LIN {X 0,Y 254.185,Z 743.005,A -85,B 0,C 180,E1 -18348.841,E2 -18348.841} C_VEL
LIN {X 0,Y 254.451,Z 743.746,A -85,B 0,C 180,E1 -18350.461,E2 -18350.461} C_VEL
LIN {X 0,Y 255.037,Z 744.003,A -85,B 0,C 180,E1 -18352.785,E2 -18352.785} C_VEL
LIN {X 0,Y 255.836,Z 743.277,A -85,B 0,C 180,E1 -18355.273,E2 -18355.273} C_VEL
LIN {X 0,Y 256.521,Z 742.248,A -85,B 0,C 180,E1 -18356.859,E2 -18356.859} C_VEL
LIN {X 0,Y 257.385,Z 740.801,A -85,B 0,C 180,E1 -18358.436,E2 -18358.436} C_VEL
LIN {X 0,Y 259.004,Z 737.791,A -85,B 0,C 180,E1 -18360.778,E2 -18360.778} C_VEL
LIN {X 0,Y 260.963,Z 733.697,A -85,B 0,C 180,E1 -18363.088,E2 -18363.088} C_VEL
LIN {X 0,Y 263.781,Z 727.398,A -85,B 0,C 180,E1 -18365.735,E2 -18365.735} C_VEL
LIN {X 0,Y 266.552,Z 720.551,A -85,B 0,C 180,E1 -18367.957,E2 -18367.957} C_VEL
LIN {X 0,Y 269.729,Z 712.054,A -85,B 0,C 180,E1 -18370.13,E2 -18370.13} C_VEL
LIN {X 0,Y 273.106,Z 701.639,A -85,B 0,C 180,E1 -18372.22,E2 -18372.22} C_VEL
LIN {X 0,Y 275.948,Z 692.039,A -85,B 0,C 180,E1 -18373.764,E2 -18373.764} C_VEL
LIN {X 0,Y 278.759,Z 681.081,A -85,B 0,C 180,E1 -18375.164,E2 -18375.164} C_VEL
LIN {X 0,Y 281.256,Z 669.518,A -85,B 0,C 180,E1 -18376.327,E2 -18376.327} C_VEL
LIN {X 0,Y 283.405,Z 656.904,A -85,B 0,C 180,E1 -18377.313,E2 -18377.313} C_VEL
LIN {X 0,Y 285.202,Z 643.24,A -85,B 0,C 180,E1 -18378.08,E2 -18378.08} C_VEL
LIN {X 0,Y 293.293,Z 569.423,A -85,B 0,C 180,E1 -18380.967,E2 -18380.967} C_VEL
LIN {X 0,Y 292.37,Z 562.086,A -85,B 0,C 180,E1 -18381.783,E2 -18381.783} C_VEL
LIN {X 0,Y 289.57,Z 555.151,A -85,B 0,C 180,E1 -18383.235,E2 -18383.235} C_VEL
LIN {X 0,Y 287.074,Z 550,A -85,B 0,C 180,E1 -18384.595,E2 -18384.595} C_VEL
LIN {X 0,Y 284.451,Z 545.04,A -85,B 0,C 180,E1 -18386.191,E2 -18386.191} C_VEL
LIN {X 0,Y 282.316,Z 541.113,A -85,B 0,C 180,E1 -18387.682,E2 -18387.682} C_VEL
LIN {X 0,Y 280.179,Z 537.278,A -85,B 0,C 180,E1 -18389.514,E2 -18389.514} C_VEL
LIN {X 0,Y 279.576,Z 534.434,A -85,B 0,C 180,E1 -18391.864,E2 -18391.864} C_VEL
LIN {X 0,Y 279.061,Z 531.769,A -85,B 0,C 180,E1 -18395.398,E2 -18395.398} C_VEL
LIN {X 0,Y 279.075,Z 531.124,A -85,B 0,C 180,E1 -18397.186,E2 -18397.186} C_VEL
LIN {X 0,Y 279.327,Z 530.927,A -85,B 0,C 180,E1 -18398.978,E2 -18398.978} C_VEL
LIN {X 0,Y 279.879,Z 531.363,A -85,B 0,C 180,E1 -18401.118,E2 -18401.118} C_VEL
LIN {X 0,Y 281.561,Z 533.211,A -85,B 0,C 180,E1 -18404.34,E2 -18404.34} C_VEL
LIN {X 0,Y 283.184,Z 535.693,A -85,B 0,C 180,E1 -18406.611,E2 -18406.611} C_VEL
LIN {X 0,Y 283.526,Z 537.108,A -85,B 0,C 180,E1 -18407.285,E2 -18407.285} C_VEL
LIN {X 0,Y 284.211,Z 543.82,A -85,B 0,C 180,E1 -18409.575,E2 -18409.575} C_VEL
LIN {X 0,Y 285.671,Z 549.141,A -85,B 0,C 180,E1 -18410.901,E2 -18410.901} C_VEL
LIN {X 0,Y 287.554,Z 555.121,A -85,B 0,C 180,E1 -18412.19,E2 -18412.19} C_VEL
LIN {X 0,Y 288.595,Z 571.291,A -85,B 0,C 180,E1 -18413.907,E2 -18413.907} C_VEL
LIN {X 0,Y 289.268,Z 589.378,A -85,B 0,C 180,E1 -18415.473,E2 -18415.473} C_VEL
LIN {X 0,Y 289.11,Z 602.402,A -85,B 0,C 180,E1 -18416.365,E2 -18416.365} C_VEL
LIN {X 0,Y 288.715,Z 612.619,A -85,B 0,C 180,E1 -18416.953,E2 -18416.953} C_VEL
LIN {X 0,Y 282.733,Z 667.61,A -85,B 0,C 180,E1 -18419.155,E2 -18419.155} C_VEL
LIN {X 0,Y 280.725,Z 680.085,A -85,B 0,C 180,E1 -18419.847,E2 -18419.847} C_VEL
LIN {X 0,Y 278.011,Z 693.453,A -85,B 0,C 180,E1 -18420.878,E2 -18420.878} C_VEL
LIN {X 0,Y 274.799,Z 706.228,A -85,B 0,C 180,E1 -18422.174,E2 -18422.174} C_VEL
LIN {X 0,Y 271.636,Z 717.557,A -85,B 0,C 180,E1 -18423.697,E2 -18423.697} C_VEL
LIN {X 0,Y 268.67,Z 727.067,A -85,B 0,C 180,E1 -18425.255,E2 -18425.255} C_VEL
LIN {X 0,Y 265.711,Z 735.889,A -85,B 0,C 180,E1 -18427.035,E2 -18427.035} C_VEL
LIN {X 0,Y 262.636,Z 744.591,A -85,B 0,C 180,E1 -18429.231,E2 -18429.231} C_VEL
LIN {X 0,Y 260.042,Z 751.709,A -85,B 0,C 180,E1 -18431.482,E2 -18431.482} C_VEL
LIN {X 0,Y 257.827,Z 758.361,A -85,B 0,C 180,E1 -18434.179,E2 -18434.179} C_VEL
LIN {X 0,Y 256.164,Z 762.774,A -85,B 0,C 180,E1 -18436.512,E2 -18436.512} C_VEL
LIN {X 0,Y 255.121,Z 766.133,A -85,B 0,C 180,E1 -18438.879,E2 -18438.879} C_VEL
LIN {X 0,Y 254.649,Z 767.83,A -85,B 0,C 180,E1 -18440.466,E2 -18440.466} C_VEL
LIN {X 0,Y 254.176,Z 769.927,A -85,B 0,C 180,E1 -18443.647,E2 -18443.647} C_VEL
LIN {X 0,Y 254.189,Z 770.373,A -85,B 0,C 180,E1 -18445.239,E2 -18445.239} C_VEL
LIN {X 0,Y 254.274,Z 770.36,A -85,B 0,C 180,E1 -18446.829,E2 -18446.829} C_VEL
LIN {X 0,Y 254.377,Z 769.902,A -85,B 0,C 180,E1 -18448.414,E2 -18448.414} C_VEL
LIN {X 0,Y 254.724,Z 769.039,A -85,B 0,C 180,E1 -18449.997,E2 -18449.997} C_VEL
LIN {X 0,Y 254.595,Z 767.669,A -85,B 0,C 180,E1 -18451.579,E2 -18451.579} C_VEL
LIN {X 0,Y 254.453,Z 764.67,A -85,B 0,C 180,E1 -18453.957,E2 -18453.957} C_VEL
LIN {X 0,Y 254.522,Z 760.49,A -85,B 0,C 180,E1 -18456.339,E2 -18456.339} C_VEL
LIN {X 0,Y 254.662,Z 754.975,A -85,B 0,C 180,E1 -18458.728,E2 -18458.728} C_VEL
LIN {X 0,Y 255.013,Z 747.964,A -85,B 0,C 180,E1 -18461.12,E2 -18461.12} C_VEL
LIN {X 0,Y 255.637,Z 740.764,A -85,B 0,C 180,E1 -18463.106,E2 -18463.106} C_VEL
LIN {X 0,Y 256.514,Z 731.989,A -85,B 0,C 180,E1 -18465.084,E2 -18465.084} C_VEL
LIN {X 0,Y 257.613,Z 720.98,A -85,B 0,C 180,E1 -18467.084,E2 -18467.084} C_VEL
LIN {X 0,Y 258.932,Z 709.068,A -85,B 0,C 180,E1 -18468.78,E2 -18468.78} C_VEL
LIN {X 0,Y 259.673,Z 701.006,A -85,B 0,C 180,E1 -18469.771,E2 -18469.771} C_VEL
LIN {X 0,Y 261.334,Z 689.069,A -85,B 0,C 180,E1 -18471.492,E2 -18471.492} C_VEL
LIN {X 0,Y 262.756,Z 679.118,A -85,B 0,C 180,E1 -18472.609,E2 -18472.609} C_VEL
LIN {X 0,Y 264.104,Z 667.499,A -85,B 0,C 180,E1 -18473.627,E2 -18473.627} C_VEL
LIN {X 0,Y 265.175,Z 654.109,A -85,B 0,C 180,E1 -18474.46,E2 -18474.46} C_VEL
LIN {X 0,Y 265.845,Z 641.126,A -85,B 0,C 180,E1 -18474.968,E2 -18474.968} C_VEL
LIN {X 0,Y 266.539,Z 604.242,A -85,B 0,C 180,E1 -18475.966,E2 -18475.966} C_VEL
LIN {X 0,Y 260.855,Z 537.989,A -85,B 0,C 180,E1 -18478.35,E2 -18478.35} C_VEL
LIN {X 0,Y 260.656,Z 535,A -85,B 0,C 180,E1 -18478.536,E2 -18478.536} C_VEL
LIN {X 0,Y 262.516,Z 522.912,A -85,B 0,C 180,E1 -18481.531,E2 -18481.531} C_VEL
LIN {X 0,Y 261.32,Z 515.677,A -85,B 0,C 180,E1 -18483.516,E2 -18483.516} C_VEL
LIN {X 0,Y 258.429,Z 502.242,A -85,B 0,C 180,E1 -18487.406,E2 -18487.406} C_VEL
LIN {X 0,Y 256.055,Z 492.707,A -85,B 0,C 180,E1 -18490.413,E2 -18490.413} C_VEL
LIN {X 0,Y 256.029,Z 492.593,A -85,B 0,C 180,E1 -18494.463,E2 -18494.463} C_VEL
LIN {X 0,Y 256.046,Z 492.591,A -85,B 0,C 180,E1 -18498.794,E2 -18498.794} C_VEL
LIN {X 0,Y 256.116,Z 492.581,A -85,B 0,C 180,E1 -18502.864,E2 -18502.864} C_VEL
LIN {X 0,Y 256.058,Z 492.587,A -85,B 0,C 180,E1 -18506.705,E2 -18506.705} C_VEL
LIN {X 0,Y 256.094,Z 492.577,A -85,B 0,C 180,E1 -18510.397,E2 -18510.397} C_VEL
LIN {X 0,Y 256.177,Z 492.573,A -85,B 0,C 180,E1 -18514.86,E2 -18514.86} C_VEL
LIN {X 0,Y 256.155,Z 492.567,A -85,B 0,C 180,E1 -18519.103,E2 -18519.103} C_VEL
LIN {X 0,Y 256.288,Z 492.56,A -85,B 0,C 180,E1 -18524.084,E2 -18524.084} C_VEL
LIN {X 0,Y 256.297,Z 492.544,A -85,B 0,C 180,E1 -18528.933,E2 -18528.933} C_VEL
LIN {X 0,Y 256.527,Z 492.527,A -85,B 0,C 180,E1 -18532.126,E2 -18532.126} C_VEL
LIN {X 0,Y 256.701,Z 492.492,A -85,B 0,C 180,E1 -18538.431,E2 -18538.431} C_VEL
LIN {X 0,Y 256.702,Z 492.503,A -85,B 0,C 180,E1 -18541.568,E2 -18541.568} C_VEL
LIN {X 0,Y 256.526,Z 492.518,A -85,B 0,C 180,E1 -18547.873,E2 -18547.873} C_VEL
LIN {X 0,Y 256.296,Z 492.553,A -85,B 0,C 180,E1 -18551.066,E2 -18551.066} C_VEL
LIN {X 0,Y 256.287,Z 492.558,A -85,B 0,C 180,E1 -18555.915,E2 -18555.915} C_VEL
LIN {X 0,Y 256.154,Z 492.566,A -85,B 0,C 180,E1 -18560.896,E2 -18560.896} C_VEL
LIN {X 0,Y 256.176,Z 492.572,A -85,B 0,C 180,E1 -18565.139,E2 -18565.139} C_VEL
LIN {X 0,Y 256.101,Z 492.572,A -85,B 0,C 180,E1 -18569.601,E2 -18569.601} C_VEL
LIN {X 0,Y 256.055,Z 492.589,A -85,B 0,C 180,E1 -18573.294,E2 -18573.294} C_VEL
LIN {X 0,Y 256.101,Z 492.571,A -85,B 0,C 180,E1 -18577.272,E2 -18577.272} C_VEL
LIN {X 0,Y 256.048,Z 492.591,A -85,B 0,C 180,E1 -18581.204,E2 -18581.204} C_VEL
LIN {X 0,Y 256.065,Z 492.583,A -85,B 0,C 180,E1 -18585.528,E2 -18585.528} C_VEL
LIN {X 0,Y 256.121,Z 492.582,A -85,B 0,C 180,E1 -18588.814,E2 -18588.814} C_VEL
LIN {X 0,Y 256.147,Z 492.549,A -85,B 0,C 180,E1 -18592.874,E2 -18592.874} C_VEL
LIN {X 0,Y 256.076,Z 492.581,A -85,B 0,C 180,E1 -18596.712,E2 -18596.712} C_VEL
LIN {X 0,Y 256.127,Z 492.562,A -85,B 0,C 180,E1 -18601.409,E2 -18601.409} C_VEL
LIN {X 0,Y 256.161,Z 492.577,A -85,B 0,C 180,E1 -18605.702,E2 -18605.702} C_VEL
LIN {X 0,Y 256.16,Z 492.565,A -85,B 0,C 180,E1 -18609.107,E2 -18609.107} C_VEL
LIN {X 0,Y 256.295,Z 492.554,A -85,B 0,C 180,E1 -18614.088,E2 -18614.088} C_VEL
LIN {X 0,Y 256.297,Z 492.78,A -85,B 0,C 180,E1 -18615.988,E2 -18615.988} C_VEL
LIN {X 0,Y 256.592,Z 493.998,A -85,B 0,C 180,E1 -18616.254,E2 -18616.254} C_VEL
LIN {X 0,Y 266.235,Z 515.857,A -85,B 0,C 180,E1 -18617.819,E2 -18617.819} C_VEL
LIN {X 0,Y 268.224,Z 521.409,A -85,B 0,C 180,E1 -18618.154,E2 -18618.154} C_VEL
LIN {X 0,Y 267.286,Z 561.383,A -85,B 0,C 180,E1 -18619.219,E2 -18619.219} C_VEL
LIN {X 0,Y 267.117,Z 579.763,A -85,B 0,C 180,E1 -18619.821,E2 -18619.821} C_VEL
LIN {X 0,Y 266.694,Z 592.285,A -85,B 0,C 180,E1 -18620.523,E2 -18620.523} C_VEL
LIN {X 0,Y 266.066,Z 603.891,A -85,B 0,C 180,E1 -18621.458,E2 -18621.458} C_VEL
LIN {X 0,Y 264.979,Z 616.183,A -85,B 0,C 180,E1 -18622.765,E2 -18622.765} C_VEL
LIN {X 0,Y 263.765,Z 627.186,A -85,B 0,C 180,E1 -18624.268,E2 -18624.268} C_VEL
LIN {X 0,Y 262.639,Z 636.11,A -85,B 0,C 180,E1 -18625.783,E2 -18625.783} C_VEL
LIN {X 0,Y 261.332,Z 645.297,A -85,B 0,C 180,E1 -18627.691,E2 -18627.691} C_VEL
LIN {X 0,Y 259.961,Z 654.232,A -85,B 0,C 180,E1 -18630.003,E2 -18630.003} C_VEL
LIN {X 0,Y 258.849,Z 661.445,A -85,B 0,C 180,E1 -18632.337,E2 -18632.337} C_VEL
LIN {X 0,Y 257.967,Z 667.219,A -85,B 0,C 180,E1 -18634.691,E2 -18634.691} C_VEL
LIN {X 0,Y 257.304,Z 671.781,A -85,B 0,C 180,E1 -18637.063,E2 -18637.063} C_VEL
LIN {X 0,Y 256.779,Z 675.721,A -85,B 0,C 180,E1 -18639.836,E2 -18639.836} C_VEL
LIN {X 0,Y 256.61,Z 678.375,A -85,B 0,C 180,E1 -18642.659,E2 -18642.659} C_VEL
LIN {X 0,Y 256.671,Z 679.326,A -85,B 0,C 180,E1 -18644.269,E2 -18644.269} C_VEL
LIN {X 0,Y 257.054,Z 679.962,A -85,B 0,C 180,E1 -18646.881,E2 -18646.881} C_VEL
LIN {X 0,Y 257.569,Z 679.652,A -85,B 0,C 180,E1 -18649.115,E2 -18649.115} C_VEL
LIN {X 0,Y 258.115,Z 678.945,A -85,B 0,C 180,E1 -18650.733,E2 -18650.733} C_VEL
LIN {X 0,Y 258.957,Z 677.506,A -85,B 0,C 180,E1 -18652.67,E2 -18652.67} C_VEL
LIN {X 0,Y 260.594,Z 674.173,A -85,B 0,C 180,E1 -18655.566,E2 -18655.566} C_VEL
LIN {X 0,Y 262.128,Z 670.526,A -85,B 0,C 180,E1 -18657.778,E2 -18657.778} C_VEL
LIN {X 0,Y 264.282,Z 664.867,A -85,B 0,C 180,E1 -18660.351,E2 -18660.351} C_VEL
LIN {X 0,Y 266.618,Z 658.1,A -85,B 0,C 180,E1 -18662.723,E2 -18662.723} C_VEL
LIN {X 0,Y 268.72,Z 651.161,A -85,B 0,C 180,E1 -18664.672,E2 -18664.672} C_VEL
LIN {X 0,Y 271.143,Z 642.643,A -85,B 0,C 180,E1 -18666.598,E2 -18666.598} C_VEL
LIN {X 0,Y 273.351,Z 633.127,A -85,B 0,C 180,E1 -18668.338,E2 -18668.338} C_VEL
LIN {X 0,Y 275.258,Z 624.075,A -85,B 0,C 180,E1 -18669.669,E2 -18669.669} C_VEL
LIN {X 0,Y 277.21,Z 612.439,A -85,B 0,C 180,E1 -18671.037,E2 -18671.037} C_VEL
LIN {X 0,Y 278.542,Z 601.085,A -85,B 0,C 180,E1 -18672.086,E2 -18672.086} C_VEL
LIN {X 0,Y 279.607,Z 588.128,A -85,B 0,C 180,E1 -18672.953,E2 -18672.953} C_VEL
LIN {X 0,Y 280.005,Z 575.71,A -85,B 0,C 180,E1 -18673.52,E2 -18673.52} C_VEL
LIN {X 0,Y 281.019,Z 538.506,A -85,B 0,C 180,E1 -18674.552,E2 -18674.552} C_VEL
LIN {X 0,Y 280.998,Z 535.255,A -85,B 0,C 180,E1 -18674.658,E2 -18674.658} C_VEL
LIN {X 0,Y 275.239,Z 524.302,A -85,B 0,C 180,E1 -18675.909,E2 -18675.909} C_VEL
LIN {X 0,Y 267.812,Z 522.35,A -85,B 0,C 180,E1 -18677.227,E2 -18677.227} C_VEL
LIN {X 0,Y 267.173,Z 522.029,A -85,B 0,C 180,E1 -18677.351,E2 -18677.351} C_VEL
LIN {X 0,Y 264.6,Z 521.929,A -85,B 0,C 180,E1 -18677.814,E2 -18677.814} C_VEL
LIN {X 0,Y 263.031,Z 520.868,A -85,B 0,C 180,E1 -18678.209,E2 -18678.209} C_VEL
LIN {X 0,Y 262.715,Z 520.837,A -85,B 0,C 180,E1 -18678.582,E2 -18678.582} C_VEL
LIN {X 0,Y 262.956,Z 522.449,A -85,B 0,C 180,E1 -18679.101,E2 -18679.101} C_VEL
LIN {X 0,Y 262.784,Z 527.936,A -85,B 0,C 180,E1 -18680.306,E2 -18680.306} C_VEL
LIN {X 0,Y 264.338,Z 542.036,A -85,B 0,C 180,E1 -18681.018,E2 -18681.018} C_VEL
LIN {X 0,Y 266.145,Z 556.491,A -85,B 0,C 180,E1 -18681.702,E2 -18681.702} C_VEL
LIN {X 0,Y 262.593,Z 640.903,A -85,B 0,C 180,E1 -18684.871,E2 -18684.871} C_VEL
LIN {X 0,Y 261.975,Z 653.038,A -85,B 0,C 180,E1 -18685.595,E2 -18685.595} C_VEL
LIN {X 0,Y 260.972,Z 666.42,A -85,B 0,C 180,E1 -18686.707,E2 -18686.707} C_VEL
LIN {X 0,Y 259.991,Z 677.997,A -85,B 0,C 180,E1 -18687.962,E2 -18687.962} C_VEL
LIN {X 0,Y 258.726,Z 690.353,A -85,B 0,C 180,E1 -18689.675,E2 -18689.675} C_VEL
LIN {X 0,Y 257.777,Z 699.276,A -85,B 0,C 180,E1 -18691.198,E2 -18691.198} C_VEL
LIN {X 0,Y 256.681,Z 703.711,A -85,B 0,C 180,E1 -18692.032,E2 -18692.032} C_VEL
LIN {X 0,Y 253.112,Z 710.462,A -85,B 0,C 180,E1 -18693.455,E2 -18693.455} C_VEL
LIN {X 0,Y 249.545,Z 716.662,A -85,B 0,C 180,E1 -18695.035,E2 -18695.035} C_VEL
LIN {X 0,Y 248.478,Z 720.238,A -85,B 0,C 180,E1 -18696.096,E2 -18696.096} C_VEL
LIN {X 0,Y 247.808,Z 726.872,A -85,B 0,C 180,E1 -18698.366,E2 -18698.366} C_VEL
LIN {X 0,Y 247.371,Z 732.842,A -85,B 0,C 180,E1 -18700.931,E2 -18700.931} C_VEL
LIN {X 0,Y 247.048,Z 737.413,A -85,B 0,C 180,E1 -18703.473,E2 -18703.473} C_VEL
LIN {X 0,Y 246.975,Z 739.992,A -85,B 0,C 180,E1 -18705.365,E2 -18705.365} C_VEL
LIN {X 0,Y 246.966,Z 741.606,A -85,B 0,C 180,E1 -18706.841,E2 -18706.841} C_VEL
LIN {X 0,Y 247.052,Z 743.005,A -85,B 0,C 180,E1 -18708.514,E2 -18708.514} C_VEL
LIN {X 0,Y 247.299,Z 743.912,A -85,B 0,C 180,E1 -18710.183,E2 -18710.183} C_VEL
LIN {X 0,Y 247.941,Z 744.475,A -85,B 0,C 180,E1 -18712.806,E2 -18712.806} C_VEL
LIN {X 0,Y 248.695,Z 744.071,A -85,B 0,C 180,E1 -18715.137,E2 -18715.137} C_VEL
LIN {X 0,Y 249.386,Z 743.272,A -85,B 0,C 180,E1 -18716.77,E2 -18716.77} C_VEL
LIN {X 0,Y 250.269,Z 742.062,A -85,B 0,C 180,E1 -18718.391,E2 -18718.391} C_VEL
LIN {X 0,Y 251.936,Z 739.373,A -85,B 0,C 180,E1 -18720.8,E2 -18720.8} C_VEL
LIN {X 0,Y 253.958,Z 735.656,A -85,B 0,C 180,E1 -18723.173,E2 -18723.173} C_VEL
LIN {X 0,Y 256.362,Z 730.805,A -85,B 0,C 180,E1 -18725.507,E2 -18725.507} C_VEL
LIN {X 0,Y 259.689,Z 723.467,A -85,B 0,C 180,E1 -18728.169,E2 -18728.169} C_VEL
LIN {X 0,Y 262.967,Z 715.568,A -85,B 0,C 180,E1 -18730.394,E2 -18730.394} C_VEL
LIN {X 0,Y 266.212,Z 706.824,A -85,B 0,C 180,E1 -18732.357,E2 -18732.357} C_VEL
LIN {X 0,Y 269.612,Z 696.708,A -85,B 0,C 180,E1 -18734.157,E2 -18734.157} C_VEL
LIN {X 0,Y 272.635,Z 685.897,A -85,B 0,C 180,E1 -18735.705,E2 -18735.705} C_VEL
LIN {X 0,Y 275.662,Z 673.866,A -85,B 0,C 180,E1 -18737.05,E2 -18737.05} C_VEL
LIN {X 0,Y 278.321,Z 660.229,A -85,B 0,C 180,E1 -18738.21,E2 -18738.21} C_VEL
LIN {X 0,Y 280.249,Z 646.973,A -85,B 0,C 180,E1 -18739.027,E2 -18739.027} C_VEL
LIN {X 0,Y 289.151,Z 571.358,A -85,B 0,C 180,E1 -18742.064,E2 -18742.064} C_VEL
LIN {X 0,Y 288.559,Z 566.13,A -85,B 0,C 180,E1 -18742.665,E2 -18742.665} C_VEL
LIN {X 0,Y 285.533,Z 558.661,A -85,B 0,C 180,E1 -18744.393,E2 -18744.393} C_VEL
LIN {X 0,Y 283.552,Z 554.334,A -85,B 0,C 180,E1 -18745.636,E2 -18745.636} C_VEL
LIN {X 0,Y 280.316,Z 547.926,A -85,B 0,C 180,E1 -18747.934,E2 -18747.934} C_VEL
LIN {X 0,Y 277.708,Z 543.218,A -85,B 0,C 180,E1 -18750.24,E2 -18750.24} C_VEL
LIN {X 0,Y 275.586,Z 539.716,A -85,B 0,C 180,E1 -18752.812,E2 -18752.812} C_VEL
LIN {X 0,Y 275.124,Z 538.444,A -85,B 0,C 180,E1 -18754.194,E2 -18754.194} C_VEL
LIN {X 0,Y 275.147,Z 537.469,A -85,B 0,C 180,E1 -18755.979,E2 -18755.979} C_VEL
LIN {X 0,Y 275.307,Z 537.019,A -85,B 0,C 180,E1 -18757.783,E2 -18757.783} C_VEL
LIN {X 0,Y 275.849,Z 537.149,A -85,B 0,C 180,E1 -18760.149,E2 -18760.149} C_VEL
LIN {X 0,Y 277.193,Z 538.507,A -85,B 0,C 180,E1 -18763.202,E2 -18763.202} C_VEL
LIN {X 0,Y 278.983,Z 540.823,A -85,B 0,C 180,E1 -18765.799,E2 -18765.799} C_VEL
LIN {X 0,Y 279.576,Z 542.512,A -85,B 0,C 180,E1 -18766.804,E2 -18766.804} C_VEL
LIN {X 0,Y 280.403,Z 546.296,A -85,B 0,C 180,E1 -18768.048,E2 -18768.048} C_VEL
LIN {X 0,Y 282.821,Z 554.731,A -85,B 0,C 180,E1 -18770.229,E2 -18770.229} C_VEL
LIN {X 0,Y 284.146,Z 559.671,A -85,B 0,C 180,E1 -18771.289,E2 -18771.289} C_VEL
LIN {X 0,Y 284.845,Z 574.82,A -85,B 0,C 180,E1 -18772.916,E2 -18772.916} C_VEL
LIN {X 0,Y 285.153,Z 592.183,A -85,B 0,C 180,E1 -18774.458,E2 -18774.458} C_VEL
LIN {X 0,Y 284.756,Z 606.968,A -85,B 0,C 180,E1 -18775.465,E2 -18775.465} C_VEL
LIN {X 0,Y 284.315,Z 614.163,A -85,B 0,C 180,E1 -18775.873,E2 -18775.873} C_VEL
LIN {X 0,Y 278.101,Z 667.643,A -85,B 0,C 180,E1 -18778.052,E2 -18778.052} C_VEL
LIN {X 0,Y 275.965,Z 679.781,A -85,B 0,C 180,E1 -18778.74,E2 -18778.74} C_VEL
LIN {X 0,Y 273.337,Z 692.001,A -85,B 0,C 180,E1 -18779.693,E2 -18779.693} C_VEL
LIN {X 0,Y 269.919,Z 704.858,A -85,B 0,C 180,E1 -18780.988,E2 -18780.988} C_VEL
LIN {X 0,Y 266.54,Z 716.406,A -85,B 0,C 180,E1 -18782.518,E2 -18782.518} C_VEL
LIN {X 0,Y 263.042,Z 726.874,A -85,B 0,C 180,E1 -18784.265,E2 -18784.265} C_VEL
LIN {X 0,Y 259.86,Z 735.565,A -85,B 0,C 180,E1 -18786.064,E2 -18786.064} C_VEL
LIN {X 0,Y 256.586,Z 744.239,A -85,B 0,C 180,E1 -18788.296,E2 -18788.296} C_VEL
LIN {X 0,Y 253.692,Z 751.31,A -85,B 0,C 180,E1 -18790.581,E2 -18790.581} C_VEL
LIN {X 0,Y 251.625,Z 757.021,A -85,B 0,C 180,E1 -18792.944,E2 -18792.944} C_VEL
LIN {X 0,Y 249.755,Z 761.624,A -85,B 0,C 180,E1 -18795.327,E2 -18795.327} C_VEL
LIN {X 0,Y 248.477,Z 765.141,A -85,B 0,C 180,E1 -18797.75,E2 -18797.75} C_VEL
LIN {X 0,Y 247.621,Z 767.671,A -85,B 0,C 180,E1 -18800.192,E2 -18800.192} C_VEL
LIN {X 0,Y 247.274,Z 768.842,A -85,B 0,C 180,E1 -18801.827,E2 -18801.827} C_VEL
LIN {X 0,Y 247.092,Z 769.865,A -85,B 0,C 180,E1 -18804.568,E2 -18804.568} C_VEL
LIN {X 0,Y 247.199,Z 769.81,A -85,B 0,C 180,E1 -18806.738,E2 -18806.738} C_VEL
LIN {X 0,Y 247.298,Z 769.284,A -85,B 0,C 180,E1 -18808.369,E2 -18808.369} C_VEL
LIN {X 0,Y 247.664,Z 768.342,A -85,B 0,C 180,E1 -18809.997,E2 -18809.997} C_VEL
LIN {X 0,Y 247.528,Z 766.846,A -85,B 0,C 180,E1 -18811.624,E2 -18811.624} C_VEL
LIN {X 0,Y 247.401,Z 763.689,A -85,B 0,C 180,E1 -18814.07,E2 -18814.07} C_VEL
LIN {X 0,Y 247.458,Z 759.332,A -85,B 0,C 180,E1 -18816.52,E2 -18816.52} C_VEL
LIN {X 0,Y 247.627,Z 753.628,A -85,B 0,C 180,E1 -18818.978,E2 -18818.978} C_VEL
LIN {X 0,Y 248.023,Z 746.35,A -85,B 0,C 180,E1 -18821.438,E2 -18821.438} C_VEL
LIN {X 0,Y 248.811,Z 737.191,A -85,B 0,C 180,E1 -18823.889,E2 -18823.889} C_VEL
LIN {X 0,Y 249.754,Z 727.715,A -85,B 0,C 180,E1 -18825.921,E2 -18825.921} C_VEL
LIN {X 0,Y 251.061,Z 715.97,A -85,B 0,C 180,E1 -18827.931,E2 -18827.931} C_VEL
LIN {X 0,Y 252.482,Z 702.692,A -85,B 0,C 180,E1 -18829.722,E2 -18829.722} C_VEL
LIN {X 0,Y 253.863,Z 692.805,A -85,B 0,C 180,E1 -18831.303,E2 -18831.303} C_VEL
LIN {X 0,Y 255.53,Z 682.258,A -85,B 0,C 180,E1 -18832.644,E2 -18832.644} C_VEL
LIN {X 0,Y 256.834,Z 671.791,A -85,B 0,C 180,E1 -18833.694,E2 -18833.694} C_VEL
LIN {X 0,Y 258.04,Z 659.09,A -85,B 0,C 180,E1 -18834.646,E2 -18834.646} C_VEL
LIN {X 0,Y 258.904,Z 646.001,A -85,B 0,C 180,E1 -18835.308,E2 -18835.308} C_VEL
LIN {X 0,Y 259.962,Z 606.035,A -85,B 0,C 180,E1 -18836.441,E2 -18836.441} C_VEL
LIN {X 0,Y 254.426,Z 540.049,A -85,B 0,C 180,E1 -18838.888,E2 -18838.888} C_VEL
LIN {X 0,Y 253.904,Z 534.255,A -85,B 0,C 180,E1 -18839.159,E2 -18839.159} C_VEL
LIN {X 0,Y 255.434,Z 524.906,A -85,B 0,C 180,E1 -18841.514,E2 -18841.514} C_VEL
LIN {X 0,Y 255.238,Z 521.387,A -85,B 0,C 180,E1 -18842.472,E2 -18842.472} C_VEL
LIN {X 0,Y 252.977,Z 510.338,A -85,B 0,C 180,E1 -18845.687,E2 -18845.687} C_VEL
LIN {X 0,Y 250.586,Z 499.877,A -85,B 0,C 180,E1 -18848.896,E2 -18848.896} C_VEL
LIN {X 0,Y 249.006,Z 493.57,A -85,B 0,C 180,E1 -18851.003,E2 -18851.003} C_VEL
LIN {X 0,Y 248.976,Z 493.472,A -85,B 0,C 180,E1 -18855.114,E2 -18855.114} C_VEL
LIN {X 0,Y 248.997,Z 493.466,A -85,B 0,C 180,E1 -18859.519,E2 -18859.519} C_VEL
LIN {X 0,Y 249.035,Z 493.464,A -85,B 0,C 180,E1 -18863.655,E2 -18863.655} C_VEL
LIN {X 0,Y 249.028,Z 493.464,A -85,B 0,C 180,E1 -18867.843,E2 -18867.843} C_VEL
LIN {X 0,Y 249.076,Z 493.446,A -85,B 0,C 180,E1 -18871.335,E2 -18871.335} C_VEL
LIN {X 0,Y 249.14,Z 493.449,A -85,B 0,C 180,E1 -18874.967,E2 -18874.967} C_VEL
LIN {X 0,Y 249.099,Z 493.443,A -85,B 0,C 180,E1 -18880.21,E2 -18880.21} C_VEL
LIN {X 0,Y 249.23,Z 493.437,A -85,B 0,C 180,E1 -18883.62,E2 -18883.62} C_VEL
LIN {X 0,Y 249.241,Z 493.422,A -85,B 0,C 180,E1 -18888.615,E2 -18888.615} C_VEL
LIN {X 0,Y 249.469,Z 493.405,A -85,B 0,C 180,E1 -18891.902,E2 -18891.902} C_VEL
LIN {X 0,Y 249.421,Z 493.405,A -85,B 0,C 180,E1 -18896.769,E2 -18896.769} C_VEL
LIN {X 0,Y 249.715,Z 493.364,A -85,B 0,C 180,E1 -18899.999,E2 -18899.999} C_VEL
LIN {X 0,Y 249.423,Z 493.413,A -85,B 0,C 180,E1 -18903.23,E2 -18903.23} C_VEL
LIN {X 0,Y 249.468,Z 493.394,A -85,B 0,C 180,E1 -18908.097,E2 -18908.097} C_VEL
LIN {X 0,Y 249.24,Z 493.432,A -85,B 0,C 180,E1 -18911.383,E2 -18911.383} C_VEL
LIN {X 0,Y 249.229,Z 493.437,A -85,B 0,C 180,E1 -18916.378,E2 -18916.378} C_VEL
LIN {X 0,Y 249.074,Z 493.452,A -85,B 0,C 180,E1 -18921.519,E2 -18921.519} C_VEL
LIN {X 0,Y 249.118,Z 493.45,A -85,B 0,C 180,E1 -18925.483,E2 -18925.483} C_VEL
LIN {X 0,Y 249.071,Z 493.444,A -85,B 0,C 180,E1 -18928.994,E2 -18928.994} C_VEL
LIN {X 0,Y 249.018,Z 493.464,A -85,B 0,C 180,E1 -18932.427,E2 -18932.427} C_VEL
LIN {X 0,Y 249.035,Z 493.456,A -85,B 0,C 180,E1 -18936.344,E2 -18936.344} C_VEL
LIN {X 0,Y 249.013,Z 493.465,A -85,B 0,C 180,E1 -18940.476,E2 -18940.476} C_VEL
LIN {X 0,Y 249.008,Z 493.458,A -85,B 0,C 180,E1 -18944.877,E2 -18944.877} C_VEL
LIN {X 0,Y 249.071,Z 493.46,A -85,B 0,C 180,E1 -18947.379,E2 -18947.379} C_VEL
LIN {X 0,Y 249.044,Z 493.445,A -85,B 0,C 180,E1 -18951.626,E2 -18951.626} C_VEL
LIN {X 0,Y 249.053,Z 493.446,A -85,B 0,C 180,E1 -18955.644,E2 -18955.644} C_VEL
LIN {X 0,Y 249.043,Z 493.46,A -85,B 0,C 180,E1 -18959.475,E2 -18959.475} C_VEL
LIN {X 0,Y 249.066,Z 493.442,A -85,B 0,C 180,E1 -18963.165,E2 -18963.165} C_VEL
LIN {X 0,Y 249.073,Z 493.455,A -85,B 0,C 180,E1 -18966.735,E2 -18966.735} C_VEL
LIN {X 0,Y 249.106,Z 493.456,A -85,B 0,C 180,E1 -18970.214,E2 -18970.214} C_VEL
LIN {X 0,Y 249.228,Z 493.437,A -85,B 0,C 180,E1 -18974.464,E2 -18974.464} C_VEL
LIN {X 0,Y 249.261,Z 493.719,A -85,B 0,C 180,E1 -18975.333,E2 -18975.333} C_VEL
LIN {X 0,Y 249.593,Z 494.99,A -85,B 0,C 180,E1 -18975.576,E2 -18975.576} C_VEL
LIN {X 0,Y 257.659,Z 512.898,A -85,B 0,C 180,E1 -18976.943,E2 -18976.943} C_VEL
LIN {X 0,Y 261.534,Z 522.459,A -85,B 0,C 180,E1 -18977.589,E2 -18977.589} C_VEL
LIN {X 0,Y 260.645,Z 565.518,A -85,B 0,C 180,E1 -18978.777,E2 -18978.777} C_VEL
LIN {X 0,Y 260.491,Z 580.939,A -85,B 0,C 180,E1 -18979.313,E2 -18979.313} C_VEL
LIN {X 0,Y 259.99,Z 594.044,A -85,B 0,C 180,E1 -18980.08,E2 -18980.08} C_VEL
LIN {X 0,Y 259.315,Z 605.456,A -85,B 0,C 180,E1 -18981.037,E2 -18981.037} C_VEL
LIN {X 0,Y 258.18,Z 617.63,A -85,B 0,C 180,E1 -18982.377,E2 -18982.377} C_VEL
LIN {X 0,Y 256.921,Z 628.535,A -85,B 0,C 180,E1 -18983.918,E2 -18983.918} C_VEL
LIN {X 0,Y 255.65,Z 638.359,A -85,B 0,C 180,E1 -18985.667,E2 -18985.667} C_VEL
LIN {X 0,Y 254.281,Z 647.325,A -85,B 0,C 180,E1 -18987.627,E2 -18987.627} C_VEL
LIN {X 0,Y 252.927,Z 656.078,A -85,B 0,C 180,E1 -18990.003,E2 -18990.003} C_VEL
LIN {X 0,Y 251.762,Z 663.106,A -85,B 0,C 180,E1 -18992.402,E2 -18992.402} C_VEL
LIN {X 0,Y 250.868,Z 668.732,A -85,B 0,C 180,E1 -18994.824,E2 -18994.824} C_VEL
LIN {X 0,Y 250.218,Z 673.175,A -85,B 0,C 180,E1 -18997.264,E2 -18997.264} C_VEL
LIN {X 0,Y 249.733,Z 676.819,A -85,B 0,C 180,E1 -18999.949,E2 -18999.949} C_VEL
LIN {X 0,Y 249.575,Z 679.561,A -85,B 0,C 180,E1 -19003.022,E2 -19003.022} C_VEL
LIN {X 0,Y 249.666,Z 680.418,A -85,B 0,C 180,E1 -19004.678,E2 -19004.678} C_VEL
LIN {X 0,Y 250.067,Z 680.955,A -85,B 0,C 180,E1 -19007.149,E2 -19007.149} C_VEL
LIN {X 0,Y 250.722,Z 680.57,A -85,B 0,C 180,E1 -19009.659,E2 -19009.659} C_VEL
LIN {X 0,Y 251.307,Z 679.77,A -85,B 0,C 180,E1 -19011.321,E2 -19011.321} C_VEL
LIN {X 0,Y 252.136,Z 678.454,A -85,B 0,C 180,E1 -19013.099,E2 -19013.099} C_VEL
LIN {X 0,Y 253.488,Z 675.896,A -85,B 0,C 180,E1 -19015.454,E2 -19015.454} C_VEL
LIN {X 0,Y 255.51,Z 671.421,A -85,B 0,C 180,E1 -19018.337,E2 -19018.337} C_VEL
LIN {X 0,Y 257.23,Z 667.194,A -85,B 0,C 180,E1 -19020.364,E2 -19020.364} C_VEL
LIN {X 0,Y 259.57,Z 660.829,A -85,B 0,C 180,E1 -19022.789,E2 -19022.789} C_VEL
LIN {X 0,Y 262.219,Z 652.712,A -85,B 0,C 180,E1 -19025.19,E2 -19025.19} C_VEL
LIN {X 0,Y 264.872,Z 643.864,A -85,B 0,C 180,E1 -19027.25,E2 -19027.25} C_VEL
LIN {X 0,Y 267.062,Z 635.002,A -85,B 0,C 180,E1 -19028.927,E2 -19028.927} C_VEL
LIN {X 0,Y 269.308,Z 624.677,A -85,B 0,C 180,E1 -19030.48,E2 -19030.48} C_VEL
LIN {X 0,Y 271.284,Z 613.463,A -85,B 0,C 180,E1 -19031.816,E2 -19031.816} C_VEL
LIN {X 0,Y 272.764,Z 601.448,A -85,B 0,C 180,E1 -19032.939,E2 -19032.939} C_VEL
LIN {X 0,Y 273.844,Z 588.508,A -85,B 0,C 180,E1 -19033.802,E2 -19033.802} C_VEL
LIN {X 0,Y 274.26,Z 575.732,A -85,B 0,C 180,E1 -19034.381,E2 -19034.381} C_VEL
LIN {X 0,Y 275.263,Z 537.702,A -85,B 0,C 180,E1 -19035.467,E2 -19035.467} C_VEL
LIN {X 0,Y 271.547,Z 530.779,A -85,B 0,C 180,E1 -19036.303,E2 -19036.303} C_VEL
LIN {X 0,Y 265.108,Z 529.188,A -85,B 0,C 180,E1 -19037.469,E2 -19037.469} C_VEL
LIN {X 0,Y 261.824,Z 528.378,A -85,B 0,C 180,E1 -19038.093,E2 -19038.093} C_VEL
LIN {X 0,Y 260.861,Z 528.174,A -85,B 0,C 180,E1 -19038.279,E2 -19038.279} C_VEL
LIN {X 0,Y 258.251,Z 528.282,A -85,B 0,C 180,E1 -19038.77,E2 -19038.77} C_VEL
LIN {X 0,Y 256.599,Z 527.354,A -85,B 0,C 180,E1 -19039.226,E2 -19039.226} C_VEL
LIN {X 0,Y 256.102,Z 527.769,A -85,B 0,C 180,E1 -19039.666,E2 -19039.666} C_VEL
LIN {X 0,Y 256.01,Z 528.833,A -85,B 0,C 180,E1 -19039.884,E2 -19039.884} C_VEL
LIN {X 0,Y 257.398,Z 542.029,A -85,B 0,C 180,E1 -19040.58,E2 -19040.58} C_VEL
LIN {X 0,Y 259.297,Z 557.377,A -85,B 0,C 180,E1 -19041.326,E2 -19041.326} C_VEL
LIN {X 0,Y 255.644,Z 640.196,A -85,B 0,C 180,E1 -19044.557,E2 -19044.557} C_VEL
LIN {X 0,Y 255.004,Z 652.711,A -85,B 0,C 180,E1 -19045.305,E2 -19045.305} C_VEL
LIN {X 0,Y 254.018,Z 665.826,A -85,B 0,C 180,E1 -19046.404,E2 -19046.404} C_VEL
LIN {X 0,Y 253.023,Z 677.486,A -85,B 0,C 180,E1 -19047.678,E2 -19047.678} C_VEL
LIN {X 0,Y 251.751,Z 689.635,A -85,B 0,C 180,E1 -19049.372,E2 -19049.372} C_VEL
LIN {X 0,Y 250.587,Z 700.75,A -85,B 0,C 180,E1 -19051.315,E2 -19051.315} C_VEL
LIN {X 0,Y 249.387,Z 711.31,A -85,B 0,C 180,E1 -19053.637,E2 -19053.637} C_VEL
LIN {X 0,Y 248.587,Z 719.29,A -85,B 0,C 180,E1 -19055.8,E2 -19055.8} C_VEL
LIN {X 0,Y 248.478,Z 720.238,A -85,B 0,C 180,E1 -19056.096,E2 -19056.096} C_VEL
LIN {X 0,Y 247.456,Z 723.644,A -85,B 0,C 180,E1 -19057.192,E2 -19057.192} C_VEL
LIN {X 0,Y 244.119,Z 728.633,A -85,B 0,C 180,E1 -19059.031,E2 -19059.031} C_VEL
LIN {X 0,Y 240.89,Z 733.003,A -85,B 0,C 180,E1 -19061.004,E2 -19061.004} C_VEL
LIN {X 0,Y 240.064,Z 735.378,A -85,B 0,C 180,E1 -19062.286,E2 -19062.286} C_VEL
LIN {X 0,Y 239.889,Z 739.833,A -85,B 0,C 180,E1 -19065.203,E2 -19065.203} C_VEL
LIN {X 0,Y 239.929,Z 742.862,A -85,B 0,C 180,E1 -19068.169,E2 -19068.169} C_VEL
LIN {X 0,Y 240.154,Z 744.01,A -85,B 0,C 180,E1 -19069.888,E2 -19069.888} C_VEL
LIN {X 0,Y 240.847,Z 744.95,A -85,B 0,C 180,E1 -19072.826,E2 -19072.826} C_VEL
LIN {X 0,Y 241.562,Z 744.794,A -85,B 0,C 180,E1 -19074.993,E2 -19074.993} C_VEL
LIN {X 0,Y 242.245,Z 744.225,A -85,B 0,C 180,E1 -19076.674,E2 -19076.674} C_VEL
LIN {X 0,Y 244.24,Z 741.736,A -85,B 0,C 180,E1 -19080.001,E2 -19080.001} C_VEL
LIN {X 0,Y 246.226,Z 738.66,A -85,B 0,C 180,E1 -19082.512,E2 -19082.512} C_VEL
LIN {X 0,Y 248.503,Z 734.668,A -85,B 0,C 180,E1 -19084.868,E2 -19084.868} C_VEL
LIN {X 0,Y 251.807,Z 728.4,A -85,B 0,C 180,E1 -19087.619,E2 -19087.619} C_VEL
LIN {X 0,Y 255.015,Z 721.601,A -85,B 0,C 180,E1 -19089.919,E2 -19089.919} C_VEL
LIN {X 0,Y 258.722,Z 713.004,A -85,B 0,C 180,E1 -19092.194,E2 -19092.194} C_VEL
LIN {X 0,Y 262.638,Z 702.643,A -85,B 0,C 180,E1 -19094.332,E2 -19094.332} C_VEL
LIN {X 0,Y 266.262,Z 691.798,A -85,B 0,C 180,E1 -19096.091,E2 -19096.091} C_VEL
LIN {X 0,Y 269.307,Z 681.08,A -85,B 0,C 180,E1 -19097.465,E2 -19097.465} C_VEL
LIN {X 0,Y 272.103,Z 669.432,A -85,B 0,C 180,E1 -19098.641,E2 -19098.641} C_VEL
LIN {X 0,Y 274.551,Z 656.71,A -85,B 0,C 180,E1 -19099.632,E2 -19099.632} C_VEL
LIN {X 0,Y 276.426,Z 643.748,A -85,B 0,C 180,E1 -19100.365,E2 -19100.365} C_VEL
LIN {X 0,Y 285.23,Z 573.222,A -85,B 0,C 180,E1 -19103.219,E2 -19103.219} C_VEL
LIN {X 0,Y 284.923,Z 570.405,A -85,B 0,C 180,E1 -19103.577,E2 -19103.577} C_VEL
LIN {X 0,Y 282.387,Z 563.68,A -85,B 0,C 180,E1 -19105.186,E2 -19105.186} C_VEL
LIN {X 0,Y 279.629,Z 557.657,A -85,B 0,C 180,E1 -19107.096,E2 -19107.096} C_VEL
LIN {X 0,Y 277.531,Z 553.319,A -85,B 0,C 180,E1 -19108.82,E2 -19108.82} C_VEL
LIN {X 0,Y 275.53,Z 549.408,A -85,B 0,C 180,E1 -19110.844,E2 -19110.844} C_VEL
LIN {X 0,Y 273.659,Z 546.099,A -85,B 0,C 180,E1 -19113.423,E2 -19113.423} C_VEL
LIN {X 0,Y 272.573,Z 543.961,A -85,B 0,C 180,E1 -19116.373,E2 -19116.373} C_VEL
LIN {X 0,Y 272.59,Z 543.451,A -85,B 0,C 180,E1 -19119.33,E2 -19119.33} C_VEL
LIN {X 0,Y 273.689,Z 544.391,A -85,B 0,C 180,E1 -19122.217,E2 -19122.217} C_VEL
LIN {X 0,Y 275.888,Z 546.776,A -85,B 0,C 180,E1 -19125.102,E2 -19125.102} C_VEL
LIN {X 0,Y 277.049,Z 548.661,A -85,B 0,C 180,E1 -19126.283,E2 -19126.283} C_VEL
LIN {X 0,Y 278.838,Z 555.635,A -85,B 0,C 180,E1 -19128.358,E2 -19128.358} C_VEL
LIN {X 0,Y 280.898,Z 563.757,A -85,B 0,C 180,E1 -19130.301,E2 -19130.301} C_VEL
LIN {X 0,Y 281.204,Z 578.68,A -85,B 0,C 180,E1 -19131.933,E2 -19131.933} C_VEL
LIN {X 0,Y 281.236,Z 595.054,A -85,B 0,C 180,E1 -19133.398,E2 -19133.398} C_VEL
LIN {X 0,Y 280.545,Z 610.158,A -85,B 0,C 180,E1 -19134.443,E2 -19134.443} C_VEL
LIN {X 0,Y 280.08,Z 615.87,A -85,B 0,C 180,E1 -19134.748,E2 -19134.748} C_VEL
LIN {X 0,Y 273.845,Z 666.33,A -85,B 0,C 180,E1 -19136.838,E2 -19136.838} C_VEL
LIN {X 0,Y 271.346,Z 679.68,A -85,B 0,C 180,E1 -19137.598,E2 -19137.598} C_VEL
LIN {X 0,Y 268.365,Z 692.669,A -85,B 0,C 180,E1 -19138.632,E2 -19138.632} C_VEL
LIN {X 0,Y 264.798,Z 705.254,A -85,B 0,C 180,E1 -19139.934,E2 -19139.934} C_VEL
LIN {X 0,Y 261.166,Z 716.478,A -85,B 0,C 180,E1 -19141.465,E2 -19141.465} C_VEL
LIN {X 0,Y 257.508,Z 726.807,A -85,B 0,C 180,E1 -19143.233,E2 -19143.233} C_VEL
LIN {X 0,Y 254.118,Z 735.449,A -85,B 0,C 180,E1 -19145.052,E2 -19145.052} C_VEL
LIN {X 0,Y 250.589,Z 743.949,A -85,B 0,C 180,E1 -19147.314,E2 -19147.314} C_VEL
LIN {X 0,Y 247.056,Z 752.019,A -85,B 0,C 180,E1 -19150.037,E2 -19150.037} C_VEL
LIN {X 0,Y 244.85,Z 757.508,A -85,B 0,C 180,E1 -19152.456,E2 -19152.456} C_VEL
LIN {X 0,Y 242.904,Z 761.857,A -85,B 0,C 180,E1 -19154.904,E2 -19154.904} C_VEL
LIN {X 0,Y 241.857,Z 764.166,A -85,B 0,C 180,E1 -19156.555,E2 -19156.555} C_VEL
LIN {X 0,Y 240.61,Z 767.54,A -85,B 0,C 180,E1 -19159.904,E2 -19159.904} C_VEL
LIN {X 0,Y 240.219,Z 768.602,A -85,B 0,C 180,E1 -19161.586,E2 -19161.586} C_VEL
LIN {X 0,Y 240.012,Z 769.447,A -85,B 0,C 180,E1 -19164.958,E2 -19164.958} C_VEL
LIN {X 0,Y 240.124,Z 769.262,A -85,B 0,C 180,E1 -19166.641,E2 -19166.641} C_VEL
LIN {X 0,Y 240.224,Z 768.629,A -85,B 0,C 180,E1 -19168.321,E2 -19168.321} C_VEL
LIN {X 0,Y 240.604,Z 767.552,A -85,B 0,C 180,E1 -19169.997,E2 -19169.997} C_VEL
LIN {X 0,Y 240.366,Z 764.987,A -85,B 0,C 180,E1 -19172.511,E2 -19172.511} C_VEL
LIN {X 0,Y 240.403,Z 761.298,A -85,B 0,C 180,E1 -19175.029,E2 -19175.029} C_VEL
LIN {X 0,Y 240.439,Z 756.324,A -85,B 0,C 180,E1 -19177.555,E2 -19177.555} C_VEL
LIN {X 0,Y 240.729,Z 749.929,A -85,B 0,C 180,E1 -19180.086,E2 -19180.086} C_VEL
LIN {X 0,Y 241.313,Z 741.769,A -85,B 0,C 180,E1 -19182.614,E2 -19182.614} C_VEL
LIN {X 0,Y 242.108,Z 733.398,A -85,B 0,C 180,E1 -19184.711,E2 -19184.711} C_VEL
LIN {X 0,Y 243.145,Z 723.134,A -85,B 0,C 180,E1 -19186.798,E2 -19186.798} C_VEL
LIN {X 0,Y 244.464,Z 711.672,A -85,B 0,C 180,E1 -19188.649,E2 -19188.649} C_VEL
LIN {X 0,Y 245.285,Z 704.219,A -85,B 0,C 180,E1 -19189.671,E2 -19189.671} C_VEL
LIN {X 0,Y 246.766,Z 693.517,A -85,B 0,C 180,E1 -19191.508,E2 -19191.508} C_VEL
LIN {X 0,Y 248.71,Z 681.77,A -85,B 0,C 180,E1 -19193.081,E2 -19193.081} C_VEL
LIN {X 0,Y 250.052,Z 671.436,A -85,B 0,C 180,E1 -19194.157,E2 -19194.157} C_VEL
LIN {X 0,Y 251.294,Z 659.018,A -85,B 0,C 180,E1 -19195.132,E2 -19195.132} C_VEL
LIN {X 0,Y 252.247,Z 645.225,A -85,B 0,C 180,E1 -19195.859,E2 -19195.859} C_VEL
LIN {X 0,Y 253.331,Z 608.294,A -85,B 0,C 180,E1 -19196.934,E2 -19196.934} C_VEL
LIN {X 0,Y 249.195,Z 555.168,A -85,B 0,C 180,E1 -19198.933,E2 -19198.933} C_VEL
LIN {X 0,Y 247.23,Z 533.219,A -85,B 0,C 180,E1 -19199.862,E2 -19199.862} C_VEL
LIN {X 0,Y 248.541,Z 525.103,A -85,B 0,C 180,E1 -19201.971,E2 -19201.971} C_VEL
LIN {X 0,Y 247.323,Z 517.635,A -85,B 0,C 180,E1 -19204.145,E2 -19204.145} C_VEL
LIN {X 0,Y 244.296,Z 503.732,A -85,B 0,C 180,E1 -19208.453,E2 -19208.453} C_VEL
LIN {X 0,Y 241.953,Z 494.444,A -85,B 0,C 180,E1 -19211.616,E2 -19211.616} C_VEL
LIN {X 0,Y 241.917,Z 494.347,A -85,B 0,C 180,E1 -19216.571,E2 -19216.571} C_VEL
LIN {X 0,Y 241.947,Z 494.341,A -85,B 0,C 180,E1 -19220.278,E2 -19220.278} C_VEL
LIN {X 0,Y 241.976,Z 494.333,A -85,B 0,C 180,E1 -19224.486,E2 -19224.486} C_VEL
LIN {X 0,Y 241.964,Z 494.346,A -85,B 0,C 180,E1 -19228.478,E2 -19228.478} C_VEL
LIN {X 0,Y 241.992,Z 494.325,A -85,B 0,C 180,E1 -19232.31,E2 -19232.31} C_VEL
LIN {X 0,Y 242.046,Z 494.334,A -85,B 0,C 180,E1 -19236.014,E2 -19236.014} C_VEL
LIN {X 0,Y 242.026,Z 494.325,A -85,B 0,C 180,E1 -19239.606,E2 -19239.606} C_VEL
LIN {X 0,Y 242.152,Z 494.319,A -85,B 0,C 180,E1 -19243.277,E2 -19243.277} C_VEL
LIN {X 0,Y 242.174,Z 494.303,A -85,B 0,C 180,E1 -19248.279,E2 -19248.279} C_VEL
LIN {X 0,Y 242.415,Z 494.283,A -85,B 0,C 180,E1 -19251.665,E2 -19251.665} C_VEL
LIN {X 0,Y 242.245,Z 494.306,A -85,B 0,C 180,E1 -19255.006,E2 -19255.006} C_VEL
LIN {X 0,Y 242.623,Z 494.244,A -85,B 0,C 180,E1 -19258.339,E2 -19258.339} C_VEL
LIN {X 0,Y 242.624,Z 494.256,A -85,B 0,C 180,E1 -19261.659,E2 -19261.659} C_VEL
LIN {X 0,Y 242.411,Z 494.277,A -85,B 0,C 180,E1 -19266.81,E2 -19266.81} C_VEL
LIN {X 0,Y 242.301,Z 494.285,A -85,B 0,C 180,E1 -19270.022,E2 -19270.022} C_VEL
LIN {X 0,Y 242.154,Z 494.319,A -85,B 0,C 180,E1 -19275.141,E2 -19275.141} C_VEL
LIN {X 0,Y 242.06,Z 494.315,A -85,B 0,C 180,E1 -19278.625,E2 -19278.625} C_VEL
LIN {X 0,Y 242,Z 494.334,A -85,B 0,C 180,E1 -19282.181,E2 -19282.181} C_VEL
LIN {X 0,Y 242.054,Z 494.329,A -85,B 0,C 180,E1 -19285.839,E2 -19285.839} C_VEL
LIN {X 0,Y 242.018,Z 494.324,A -85,B 0,C 180,E1 -19289.581,E2 -19289.581} C_VEL
LIN {X 0,Y 241.968,Z 494.343,A -85,B 0,C 180,E1 -19293.494,E2 -19293.494} C_VEL
LIN {X 0,Y 241.977,Z 494.329,A -85,B 0,C 180,E1 -19297.583,E2 -19297.583} C_VEL
LIN {X 0,Y 241.936,Z 494.347,A -85,B 0,C 180,E1 -19301.922,E2 -19301.922} C_VEL
LIN {X 0,Y 241.991,Z 494.337,A -85,B 0,C 180,E1 -19306.556,E2 -19306.556} C_VEL
LIN {X 0,Y 242.001,Z 494.333,A -85,B 0,C 180,E1 -19310.294,E2 -19310.294} C_VEL
LIN {X 0,Y 242.028,Z 494.305,A -85,B 0,C 180,E1 -19314.5,E2 -19314.5} C_VEL
LIN {X 0,Y 241.968,Z 494.345,A -85,B 0,C 180,E1 -19318.482,E2 -19318.482} C_VEL
LIN {X 0,Y 241.999,Z 494.317,A -85,B 0,C 180,E1 -19322.315,E2 -19322.315} C_VEL
LIN {X 0,Y 242.051,Z 494.334,A -85,B 0,C 180,E1 -19326.019,E2 -19326.019} C_VEL
LIN {X 0,Y 242.032,Z 494.328,A -85,B 0,C 180,E1 -19329.611,E2 -19329.611} C_VEL
LIN {X 0,Y 242.213,Z 494.397,A -85,B 0,C 180,E1 -19334.459,E2 -19334.459} C_VEL
LIN {X 0,Y 242.394,Z 495.365,A -85,B 0,C 180,E1 -19334.798,E2 -19334.798} C_VEL
LIN {X 0,Y 251.281,Z 515.138,A -85,B 0,C 180,E1 -19336.388,E2 -19336.388} C_VEL
LIN {X 0,Y 254.9,Z 523.936,A -85,B 0,C 180,E1 -19337.013,E2 -19337.013} C_VEL
LIN {X 0,Y 254.037,Z 569.18,A -85,B 0,C 180,E1 -19338.304,E2 -19338.304} C_VEL
LIN {X 0,Y 253.886,Z 583.062,A -85,B 0,C 180,E1 -19338.83,E2 -19338.83} C_VEL
LIN {X 0,Y 253.299,Z 595.709,A -85,B 0,C 180,E1 -19339.613,E2 -19339.613} C_VEL
LIN {X 0,Y 252.416,Z 608.917,A -85,B 0,C 180,E1 -19340.79,E2 -19340.79} C_VEL
LIN {X 0,Y 251.283,Z 620.517,A -85,B 0,C 180,E1 -19342.166,E2 -19342.166} C_VEL
LIN {X 0,Y 249.754,Z 632.169,A -85,B 0,C 180,E1 -19343.945,E2 -19343.945} C_VEL
LIN {X 0,Y 248.347,Z 642.497,A -85,B 0,C 180,E1 -19345.946,E2 -19345.946} C_VEL
LIN {X 0,Y 246.993,Z 650.899,A -85,B 0,C 180,E1 -19347.964,E2 -19347.964} C_VEL
LIN {X 0,Y 245.66,Z 659.101,A -85,B 0,C 180,E1 -19350.413,E2 -19350.413} C_VEL
LIN {X 0,Y 244.659,Z 664.736,A -85,B 0,C 180,E1 -19352.472,E2 -19352.472} C_VEL
LIN {X 0,Y 243.752,Z 670.24,A -85,B 0,C 180,E1 -19354.965,E2 -19354.965} C_VEL
LIN {X 0,Y 243.111,Z 674.57,A -85,B 0,C 180,E1 -19357.477,E2 -19357.477} C_VEL
LIN {X 0,Y 242.674,Z 677.896,A -85,B 0,C 180,E1 -19360.052,E2 -19360.052} C_VEL
LIN {X 0,Y 242.559,Z 679.496,A -85,B 0,C 180,E1 -19361.705,E2 -19361.705} C_VEL
LIN {X 0,Y 242.564,Z 680.713,A -85,B 0,C 180,E1 -19363.405,E2 -19363.405} C_VEL
LIN {X 0,Y 242.991,Z 681.886,A -85,B 0,C 180,E1 -19366.815,E2 -19366.815} C_VEL
LIN {X 0,Y 243.353,Z 681.897,A -85,B 0,C 180,E1 -19368.525,E2 -19368.525} C_VEL
LIN {X 0,Y 243.874,Z 681.454,A -85,B 0,C 180,E1 -19370.234,E2 -19370.234} C_VEL
LIN {X 0,Y 245.34,Z 679.399,A -85,B 0,C 180,E1 -19373.557,E2 -19373.557} C_VEL
LIN {X 0,Y 246.898,Z 676.564,A -85,B 0,C 180,E1 -19376.184,E2 -19376.184} C_VEL
LIN {X 0,Y 248.924,Z 672.309,A -85,B 0,C 180,E1 -19378.928,E2 -19378.928} C_VEL
LIN {X 0,Y 251.299,Z 666.591,A -85,B 0,C 180,E1 -19381.629,E2 -19381.629} C_VEL
LIN {X 0,Y 253.844,Z 659.92,A -85,B 0,C 180,E1 -19384.055,E2 -19384.055} C_VEL
LIN {X 0,Y 256.257,Z 652.754,A -85,B 0,C 180,E1 -19386.135,E2 -19386.135} C_VEL
LIN {X 0,Y 258.769,Z 644.62,A -85,B 0,C 180,E1 -19388.037,E2 -19388.037} C_VEL
LIN {X 0,Y 261.063,Z 635.686,A -85,B 0,C 180,E1 -19389.748,E2 -19389.748} C_VEL
LIN {X 0,Y 263.427,Z 625.283,A -85,B 0,C 180,E1 -19391.326,E2 -19391.326} C_VEL
LIN {X 0,Y 265.573,Z 613.295,A -85,B 0,C 180,E1 -19392.765,E2 -19392.765} C_VEL
LIN {X 0,Y 267.053,Z 601.361,A -85,B 0,C 180,E1 -19393.869,E2 -19393.869} C_VEL
LIN {X 0,Y 268.162,Z 588.293,A -85,B 0,C 180,E1 -19394.727,E2 -19394.727} C_VEL
LIN {X 0,Y 268.569,Z 576.005,A -85,B 0,C 180,E1 -19395.276,E2 -19395.276} C_VEL
LIN {X 0,Y 269.579,Z 540.187,A -85,B 0,C 180,E1 -19396.316,E2 -19396.316} C_VEL
LIN {X 0,Y 268.002,Z 537.078,A -85,B 0,C 180,E1 -19396.69,E2 -19396.69} C_VEL
LIN {X 0,Y 259.552,Z 535.364,A -85,B 0,C 180,E1 -19398.265,E2 -19398.265} C_VEL
LIN {X 0,Y 257.483,Z 535.446,A -85,B 0,C 180,E1 -19398.655,E2 -19398.655} C_VEL
LIN {X 0,Y 255.479,Z 539.89,A -85,B 0,C 180,E1 -19398.881,E2 -19398.881} C_VEL
LIN {X 0,Y 253.787,Z 541.917,A -85,B 0,C 180,E1 -19399.139,E2 -19399.139} C_VEL
LIN {X 0,Y 253.093,Z 542.228,A -85,B 0,C 180,E1 -19399.266,E2 -19399.266} C_VEL
LIN {X 0,Y 251.312,Z 542.28,A -85,B 0,C 180,E1 -19399.698,E2 -19399.698} C_VEL
LIN {X 0,Y 250.898,Z 543.696,A -85,B 0,C 180,E1 -19400.059,E2 -19400.059} C_VEL
LIN {X 0,Y 251.092,Z 547.459,A -85,B 0,C 180,E1 -19400.412,E2 -19400.412} C_VEL
LIN {X 0,Y 252.407,Z 558.188,A -85,B 0,C 180,E1 -19400.962,E2 -19400.962} C_VEL
LIN {X 0,Y 248.63,Z 641.159,A -85,B 0,C 180,E1 -19404.311,E2 -19404.311} C_VEL
LIN {X 0,Y 247.916,Z 654.138,A -85,B 0,C 180,E1 -19405.129,E2 -19405.129} C_VEL
LIN {X 0,Y 246.847,Z 668.395,A -85,B 0,C 180,E1 -19406.4,E2 -19406.4} C_VEL
LIN {X 0,Y 245.706,Z 680.327,A -85,B 0,C 180,E1 -19407.81,E2 -19407.81} C_VEL
LIN {X 0,Y 244.416,Z 692.416,A -85,B 0,C 180,E1 -19409.618,E2 -19409.618} C_VEL
LIN {X 0,Y 243.199,Z 703.66,A -85,B 0,C 180,E1 -19411.758,E2 -19411.758} C_VEL
LIN {X 0,Y 242.22,Z 712.338,A -85,B 0,C 180,E1 -19413.785,E2 -19413.785} C_VEL
LIN {X 0,Y 241.42,Z 720.048,A -85,B 0,C 180,E1 -19415.973,E2 -19415.973} C_VEL
LIN {X 0,Y 240.664,Z 727.405,A -85,B 0,C 180,E1 -19418.562,E2 -19418.562} C_VEL
LIN {X 0,Y 240.203,Z 733.417,A -85,B 0,C 180,E1 -19421.226,E2 -19421.226} C_VEL
LIN {X 0,Y 240.064,Z 735.378,A -85,B 0,C 180,E1 -19422.286,E2 -19422.286} C_VEL
LIN {X 0,Y 239.272,Z 737.557,A -85,B 0,C 180,E1 -19423.588,E2 -19423.588} C_VEL
LIN {X 0,Y 236.288,Z 740.493,A -85,B 0,C 180,E1 -19425.755,E2 -19425.755} C_VEL
LIN {X 0,Y 233.902,Z 742.383,A -85,B 0,C 180,E1 -19427.555,E2 -19427.555} C_VEL
LIN {X 0,Y 232.998,Z 743.557,A -85,B 0,C 180,E1 -19428.966,E2 -19428.966} C_VEL
LIN {X 0,Y 232.984,Z 743.885,A -85,B 0,C 180,E1 -19429.444,E2 -19429.444} C_VEL
LIN {X 0,Y 233.35,Z 744.884,A -85,B 0,C 180,E1 -19431.34,E2 -19431.34} C_VEL
LIN {X 0,Y 233.823,Z 745.373,A -85,B 0,C 180,E1 -19433.095,E2 -19433.095} C_VEL
LIN {X 0,Y 234.41,Z 745.429,A -85,B 0,C 180,E1 -19434.84,E2 -19434.84} C_VEL
LIN {X 0,Y 235.093,Z 745.043,A -85,B 0,C 180,E1 -19436.573,E2 -19436.573} C_VEL
LIN {X 0,Y 236.028,Z 744.249,A -85,B 0,C 180,E1 -19438.294,E2 -19438.294} C_VEL
LIN {X 0,Y 237.14,Z 743.049,A -85,B 0,C 180,E1 -19440.001,E2 -19440.001} C_VEL
LIN {X 0,Y 239.212,Z 740.274,A -85,B 0,C 180,E1 -19442.621,E2 -19442.621} C_VEL
LIN {X 0,Y 242.4,Z 735.236,A -85,B 0,C 180,E1 -19445.825,E2 -19445.825} C_VEL
LIN {X 0,Y 246.001,Z 729.013,A -85,B 0,C 180,E1 -19448.627,E2 -19448.627} C_VEL
LIN {X 0,Y 249.424,Z 722.205,A -85,B 0,C 180,E1 -19450.965,E2 -19450.965} C_VEL
LIN {X 0,Y 253.338,Z 713.845,A -85,B 0,C 180,E1 -19453.242,E2 -19453.242} C_VEL
LIN {X 0,Y 256.803,Z 705.398,A -85,B 0,C 180,E1 -19455.07,E2 -19455.07} C_VEL
LIN {X 0,Y 260.995,Z 693.847,A -85,B 0,C 180,E1 -19457.029,E2 -19457.029} C_VEL
LIN {X 0,Y 264.207,Z 683.62,A -85,B 0,C 180,E1 -19458.415,E2 -19458.415} C_VEL
LIN {X 0,Y 267.59,Z 670.794,A -85,B 0,C 180,E1 -19459.765,E2 -19459.765} C_VEL
LIN {X 0,Y 270.143,Z 658.351,A -85,B 0,C 180,E1 -19460.761,E2 -19460.761} C_VEL
LIN {X 0,Y 272.272,Z 644.641,A -85,B 0,C 180,E1 -19461.553,E2 -19461.553} C_VEL
LIN {X 0,Y 281.521,Z 575.23,A -85,B 0,C 180,E1 -19464.399,E2 -19464.399} C_VEL
LIN {X 0,Y 279.457,Z 569.101,A -85,B 0,C 180,E1 -19465.908,E2 -19465.908} C_VEL
LIN {X 0,Y 277.001,Z 563.348,A -85,B 0,C 180,E1 -19467.803,E2 -19467.803} C_VEL
LIN {X 0,Y 275.329,Z 559.642,A -85,B 0,C 180,E1 -19469.308,E2 -19469.308} C_VEL
LIN {X 0,Y 273.636,Z 556.096,A -85,B 0,C 180,E1 -19471.151,E2 -19471.151} C_VEL
LIN {X 0,Y 271.907,Z 552.705,A -85,B 0,C 180,E1 -19473.826,E2 -19473.826} C_VEL
LIN {X 0,Y 271.025,Z 550.829,A -85,B 0,C 180,E1 -19476.614,E2 -19476.614} C_VEL
LIN {X 0,Y 271.002,Z 550.383,A -85,B 0,C 180,E1 -19478.919,E2 -19478.919} C_VEL
LIN {X 0,Y 271.747,Z 550.919,A -85,B 0,C 180,E1 -19481.406,E2 -19481.406} C_VEL
LIN {X 0,Y 273.212,Z 552.556,A -85,B 0,C 180,E1 -19483.802,E2 -19483.802} C_VEL
LIN {X 0,Y 274.538,Z 554.26,A -85,B 0,C 180,E1 -19485.36,E2 -19485.36} C_VEL
LIN {X 0,Y 275.093,Z 555.837,A -85,B 0,C 180,E1 -19486.032,E2 -19486.032} C_VEL
LIN {X 0,Y 276.542,Z 562.46,A -85,B 0,C 180,E1 -19487.945,E2 -19487.945} C_VEL
LIN {X 0,Y 277.765,Z 568.286,A -85,B 0,C 180,E1 -19489.34,E2 -19489.34} C_VEL
LIN {X 0,Y 277.779,Z 583.037,A -85,B 0,C 180,E1 -19490.942,E2 -19490.942} C_VEL
LIN {X 0,Y 277.463,Z 597.771,A -85,B 0,C 180,E1 -19492.281,E2 -19492.281} C_VEL
LIN {X 0,Y 276.541,Z 614.204,A -85,B 0,C 180,E1 -19493.424,E2 -19493.424} C_VEL
LIN {X 0,Y 269.618,Z 666.468,A -85,B 0,C 180,E1 -19495.63,E2 -19495.63} C_VEL
LIN {X 0,Y 266.885,Z 680.152,A -85,B 0,C 180,E1 -19496.424,E2 -19496.424} C_VEL
LIN {X 0,Y 263.512,Z 693.554,A -85,B 0,C 180,E1 -19497.535,E2 -19497.535} C_VEL
LIN {X 0,Y 259.767,Z 705.672,A -85,B 0,C 180,E1 -19498.837,E2 -19498.837} C_VEL
LIN {X 0,Y 255.968,Z 716.76,A -85,B 0,C 180,E1 -19500.379,E2 -19500.379} C_VEL
LIN {X 0,Y 252.098,Z 726.909,A -85,B 0,C 180,E1 -19502.16,E2 -19502.16} C_VEL
LIN {X 0,Y 247.815,Z 736.827,A -85,B 0,C 180,E1 -19504.372,E2 -19504.372} C_VEL
LIN {X 0,Y 244.13,Z 745.038,A -85,B 0,C 180,E1 -19506.679,E2 -19506.679} C_VEL
LIN {X 0,Y 241.052,Z 751.504,A -85,B 0,C 180,E1 -19508.971,E2 -19508.971} C_VEL
LIN {X 0,Y 238.098,Z 757.906,A -85,B 0,C 180,E1 -19511.942,E2 -19511.942} C_VEL
LIN {X 0,Y 236.054,Z 762.056,A -85,B 0,C 180,E1 -19514.455,E2 -19514.455} C_VEL
LIN {X 0,Y 234.927,Z 764.248,A -85,B 0,C 180,E1 -19516.15,E2 -19516.15} C_VEL
LIN {X 0,Y 234.179,Z 766.027,A -85,B 0,C 180,E1 -19517.87,E2 -19517.87} C_VEL
LIN {X 0,Y 233.585,Z 767.369,A -85,B 0,C 180,E1 -19519.597,E2 -19519.597} C_VEL
LIN {X 0,Y 232.968,Z 768.833,A -85,B 0,C 180,E1 -19523.066,E2 -19523.066} C_VEL
LIN {X 0,Y 232.952,Z 768.971,A -85,B 0,C 180,E1 -19524.804,E2 -19524.804} C_VEL
LIN {X 0,Y 233.051,Z 768.665,A -85,B 0,C 180,E1 -19526.539,E2 -19526.539} C_VEL
LIN {X 0,Y 233.155,Z 767.919,A -85,B 0,C 180,E1 -19528.27,E2 -19528.27} C_VEL
LIN {X 0,Y 233.545,Z 766.761,A -85,B 0,C 180,E1 -19529.997,E2 -19529.997} C_VEL
LIN {X 0,Y 233.329,Z 764.026,A -85,B 0,C 180,E1 -19532.587,E2 -19532.587} C_VEL
LIN {X 0,Y 233.359,Z 760.149,A -85,B 0,C 180,E1 -19535.181,E2 -19535.181} C_VEL
LIN {X 0,Y 233.425,Z 754.968,A -85,B 0,C 180,E1 -19537.784,E2 -19537.784} C_VEL
LIN {X 0,Y 233.727,Z 748.279,A -85,B 0,C 180,E1 -19540.391,E2 -19540.391} C_VEL
LIN {X 0,Y 234.375,Z 739.885,A -85,B 0,C 180,E1 -19542.994,E2 -19542.994} C_VEL
LIN {X 0,Y 235.239,Z 731.231,A -85,B 0,C 180,E1 -19545.151,E2 -19545.151} C_VEL
LIN {X 0,Y 236.339,Z 720.556,A -85,B 0,C 180,E1 -19547.296,E2 -19547.296} C_VEL
LIN {X 0,Y 237.55,Z 710.106,A -85,B 0,C 180,E1 -19548.989,E2 -19548.989} C_VEL
LIN {X 0,Y 238.192,Z 704.587,A -85,B 0,C 180,E1 -19549.832,E2 -19549.832} C_VEL
LIN {X 0,Y 239.672,Z 694.222,A -85,B 0,C 180,E1 -19551.725,E2 -19551.725} C_VEL
LIN {X 0,Y 241.646,Z 682.849,A -85,B 0,C 180,E1 -19553.342,E2 -19553.342} C_VEL
LIN {X 0,Y 243.134,Z 672.027,A -85,B 0,C 180,E1 -19554.549,E2 -19554.549} C_VEL
LIN {X 0,Y 244.41,Z 660.267,A -85,B 0,C 180,E1 -19555.548,E2 -19555.548} C_VEL
LIN {X 0,Y 245.421,Z 647.811,A -85,B 0,C 180,E1 -19556.29,E2 -19556.29} C_VEL
LIN {X 0,Y 246.069,Z 631.92,A -85,B 0,C 180,E1 -19556.844,E2 -19556.844} C_VEL
LIN {X 0,Y 246.601,Z 606.172,A -85,B 0,C 180,E1 -19557.594,E2 -19557.594} C_VEL
LIN {X 0,Y 241.532,Z 542.739,A -85,B 0,C 180,E1 -19560.097,E2 -19560.097} C_VEL
LIN {X 0,Y 240.549,Z 532.288,A -85,B 0,C 180,E1 -19560.591,E2 -19560.591} C_VEL
LIN {X 0,Y 241.595,Z 526.144,A -85,B 0,C 180,E1 -19562.218,E2 -19562.218} C_VEL
LIN {X 0,Y 240.029,Z 517.188,A -85,B 0,C 180,E1 -19564.931,E2 -19564.931} C_VEL
LIN {X 0,Y 237.383,Z 505.282,A -85,B 0,C 180,E1 -19568.754,E2 -19568.754} C_VEL
LIN {X 0,Y 234.894,Z 495.326,A -85,B 0,C 180,E1 -19572.261,E2 -19572.261} C_VEL
LIN {X 0,Y 234.87,Z 495.224,A -85,B 0,C 180,E1 -19576.509,E2 -19576.509} C_VEL
LIN {X 0,Y 234.909,Z 495.22,A -85,B 0,C 180,E1 -19581.076,E2 -19581.076} C_VEL
LIN {X 0,Y 234.919,Z 495.209,A -85,B 0,C 180,E1 -19585.359,E2 -19585.359} C_VEL
LIN {X 0,Y 234.913,Z 495.221,A -85,B 0,C 180,E1 -19589.429,E2 -19589.429} C_VEL
LIN {X 0,Y 234.983,Z 495.205,A -85,B 0,C 180,E1 -19593.792,E2 -19593.792} C_VEL
LIN {X 0,Y 235,Z 495.201,A -85,B 0,C 180,E1 -19598.968,E2 -19598.968} C_VEL
LIN {X 0,Y 235.085,Z 495.2,A -85,B 0,C 180,E1 -19603.058,E2 -19603.058} C_VEL
LIN {X 0,Y 235.135,Z 495.181,A -85,B 0,C 180,E1 -19607.922,E2 -19607.922} C_VEL
LIN {X 0,Y 235.364,Z 495.161,A -85,B 0,C 180,E1 -19611.413,E2 -19611.413} C_VEL
LIN {X 0,Y 235.391,Z 495.162,A -85,B 0,C 180,E1 -19613.14,E2 -19613.14} C_VEL
LIN {X 0,Y 235.582,Z 495.119,A -85,B 0,C 180,E1 -19618.29,E2 -19618.29} C_VEL
LIN {X 0,Y 235.583,Z 495.133,A -85,B 0,C 180,E1 -19621.709,E2 -19621.709} C_VEL
LIN {X 0,Y 235.391,Z 495.151,A -85,B 0,C 180,E1 -19626.858,E2 -19626.858} C_VEL
LIN {X 0,Y 235.225,Z 495.167,A -85,B 0,C 180,E1 -19630.326,E2 -19630.326} C_VEL
LIN {X 0,Y 235.101,Z 495.196,A -85,B 0,C 180,E1 -19635.607,E2 -19635.607} C_VEL
LIN {X 0,Y 234.996,Z 495.191,A -85,B 0,C 180,E1 -19639.206,E2 -19639.206} C_VEL
LIN {X 0,Y 234.948,Z 495.217,A -85,B 0,C 180,E1 -19642.883,E2 -19642.883} C_VEL
LIN {X 0,Y 234.957,Z 495.21,A -85,B 0,C 180,E1 -19646.658,E2 -19646.658} C_VEL
LIN {X 0,Y 234.919,Z 495.211,A -85,B 0,C 180,E1 -19650.569,E2 -19650.569} C_VEL
LIN {X 0,Y 234.918,Z 495.221,A -85,B 0,C 180,E1 -19654.639,E2 -19654.639} C_VEL
LIN {X 0,Y 234.93,Z 495.212,A -85,B 0,C 180,E1 -19658.946,E2 -19658.946} C_VEL
LIN {X 0,Y 234.911,Z 495.215,A -85,B 0,C 180,E1 -19663.479,E2 -19663.479} C_VEL
LIN {X 0,Y 234.964,Z 495.212,A -85,B 0,C 180,E1 -19666.536,E2 -19666.536} C_VEL
LIN {X 0,Y 234.945,Z 495.202,A -85,B 0,C 180,E1 -19671.088,E2 -19671.088} C_VEL
LIN {X 0,Y 234.952,Z 495.194,A -85,B 0,C 180,E1 -19675.369,E2 -19675.369} C_VEL
LIN {X 0,Y 234.961,Z 495.209,A -85,B 0,C 180,E1 -19680.16,E2 -19680.16} C_VEL
LIN {X 0,Y 234.987,Z 495.199,A -85,B 0,C 180,E1 -19683.796,E2 -19683.796} C_VEL
LIN {X 0,Y 235.006,Z 495.197,A -85,B 0,C 180,E1 -19688.973,E2 -19688.973} C_VEL
LIN {X 0,Y 235.15,Z 495.332,A -85,B 0,C 180,E1 -19693.706,E2 -19693.706} C_VEL
LIN {X 0,Y 235.397,Z 496.297,A -85,B 0,C 180,E1 -19694.027,E2 -19694.027} C_VEL
LIN {X 0,Y 244.085,Z 515.336,A -85,B 0,C 180,E1 -19695.65,E2 -19695.65} C_VEL
LIN {X 0,Y 248.426,Z 526.02,A -85,B 0,C 180,E1 -19696.44,E2 -19696.44} C_VEL
LIN {X 0,Y 247.448,Z 568.967,A -85,B 0,C 180,E1 -19697.686,E2 -19697.686} C_VEL
LIN {X 0,Y 247.293,Z 582.635,A -85,B 0,C 180,E1 -19698.195,E2 -19698.195} C_VEL
LIN {X 0,Y 246.77,Z 594.775,A -85,B 0,C 180,E1 -19698.919,E2 -19698.919} C_VEL
LIN {X 0,Y 246.033,Z 606.517,A -85,B 0,C 180,E1 -19699.926,E2 -19699.926} C_VEL
LIN {X 0,Y 244.839,Z 618.854,A -85,B 0,C 180,E1 -19701.335,E2 -19701.335} C_VEL
LIN {X 0,Y 243.44,Z 629.918,A -85,B 0,C 180,E1 -19702.955,E2 -19702.955} C_VEL
LIN {X 0,Y 242.186,Z 638.875,A -85,B 0,C 180,E1 -19704.591,E2 -19704.591} C_VEL
LIN {X 0,Y 240.712,Z 648.103,A -85,B 0,C 180,E1 -19706.655,E2 -19706.655} C_VEL
LIN {X 0,Y 239.276,Z 656.533,A -85,B 0,C 180,E1 -19708.997,E2 -19708.997} C_VEL
LIN {X 0,Y 237.953,Z 664.296,A -85,B 0,C 180,E1 -19711.695,E2 -19711.695} C_VEL
LIN {X 0,Y 236.956,Z 670.1,A -85,B 0,C 180,E1 -19714.255,E2 -19714.255} C_VEL
LIN {X 0,Y 236.193,Z 674.691,A -85,B 0,C 180,E1 -19716.838,E2 -19716.838} C_VEL
LIN {X 0,Y 235.628,Z 678.986,A -85,B 0,C 180,E1 -19720.176,E2 -19720.176} C_VEL
LIN {X 0,Y 235.526,Z 680.715,A -85,B 0,C 180,E1 -19722.059,E2 -19722.059} C_VEL
LIN {X 0,Y 235.553,Z 681.842,A -85,B 0,C 180,E1 -19723.812,E2 -19723.812} C_VEL
LIN {X 0,Y 236.052,Z 682.921,A -85,B 0,C 180,E1 -19727.324,E2 -19727.324} C_VEL
LIN {X 0,Y 236.464,Z 682.843,A -85,B 0,C 180,E1 -19729.086,E2 -19729.086} C_VEL
LIN {X 0,Y 237.052,Z 682.335,A -85,B 0,C 180,E1 -19730.844,E2 -19730.844} C_VEL
LIN {X 0,Y 238.539,Z 680.357,A -85,B 0,C 180,E1 -19734.03,E2 -19734.03} C_VEL
LIN {X 0,Y 240.331,Z 677.219,A -85,B 0,C 180,E1 -19736.956,E2 -19736.956} C_VEL
LIN {X 0,Y 242.342,Z 673.218,A -85,B 0,C 180,E1 -19739.541,E2 -19739.541} C_VEL
LIN {X 0,Y 245.08,Z 666.949,A -85,B 0,C 180,E1 -19742.529,E2 -19742.529} C_VEL
LIN {X 0,Y 247.832,Z 660.002,A -85,B 0,C 180,E1 -19745.05,E2 -19745.05} C_VEL
LIN {X 0,Y 250.367,Z 652.777,A -85,B 0,C 180,E1 -19747.126,E2 -19747.126} C_VEL
LIN {X 0,Y 253.296,Z 643.139,A -85,B 0,C 180,E1 -19749.333,E2 -19749.333} C_VEL
LIN {X 0,Y 255.999,Z 632.76,A -85,B 0,C 180,E1 -19751.217,E2 -19751.217} C_VEL
LIN {X 0,Y 258.543,Z 621.31,A -85,B 0,C 180,E1 -19752.814,E2 -19752.814} C_VEL
LIN {X 0,Y 260.506,Z 609.239,A -85,B 0,C 180,E1 -19754.14,E2 -19754.14} C_VEL
LIN {X 0,Y 261.815,Z 598.132,A -85,B 0,C 180,E1 -19755.066,E2 -19755.066} C_VEL
LIN {X 0,Y 262.656,Z 585.533,A -85,B 0,C 180,E1 -19755.83,E2 -19755.83} C_VEL
LIN {X 0,Y 263.092,Z 570.143,A -85,B 0,C 180,E1 -19756.4,E2 -19756.4} C_VEL
LIN {X 0,Y 263.959,Z 543.476,A -85,B 0,C 180,E1 -19757.175,E2 -19757.175} C_VEL
LIN {X 0,Y 260.11,Z 542.946,A -85,B 0,C 180,E1 -19757.889,E2 -19757.889} C_VEL
LIN {X 0,Y 257.398,Z 546.753,A -85,B 0,C 180,E1 -19758.259,E2 -19758.259} C_VEL
LIN {X 0,Y 254.816,Z 548.677,A -85,B 0,C 180,E1 -19758.685,E2 -19758.685} C_VEL
LIN {X 0,Y 253.433,Z 549.17,A -85,B 0,C 180,E1 -19758.938,E2 -19758.938} C_VEL
LIN {X 0,Y 251.218,Z 554.972,A -85,B 0,C 180,E1 -19759.162,E2 -19759.162} C_VEL
LIN {X 0,Y 249.29,Z 557.798,A -85,B 0,C 180,E1 -19759.446,E2 -19759.446} C_VEL
LIN {X 0,Y 248.209,Z 558.523,A -85,B 0,C 180,E1 -19759.64,E2 -19759.64} C_VEL
LIN {X 0,Y 246.403,Z 558.527,A -85,B 0,C 180,E1 -19760.1,E2 -19760.1} C_VEL
LIN {X 0,Y 245.61,Z 561.571,A -85,B 0,C 180,E1 -19760.526,E2 -19760.526} C_VEL
LIN {X 0,Y 245.13,Z 567.114,A -85,B 0,C 180,E1 -19760.895,E2 -19760.895} C_VEL
LIN {X 0,Y 241.63,Z 641.901,A -85,B 0,C 180,E1 -19764.044,E2 -19764.044} C_VEL
LIN {X 0,Y 240.85,Z 655.066,A -85,B 0,C 180,E1 -19764.919,E2 -19764.919} C_VEL
LIN {X 0,Y 239.835,Z 668.56,A -85,B 0,C 180,E1 -19766.168,E2 -19766.168} C_VEL
LIN {X 0,Y 238.55,Z 681.267,A -85,B 0,C 180,E1 -19767.726,E2 -19767.726} C_VEL
LIN {X 0,Y 237.322,Z 692.666,A -85,B 0,C 180,E1 -19769.494,E2 -19769.494} C_VEL
LIN {X 0,Y 236.158,Z 703.322,A -85,B 0,C 180,E1 -19771.566,E2 -19771.566} C_VEL
LIN {X 0,Y 235.061,Z 713.132,A -85,B 0,C 180,E1 -19773.912,E2 -19773.912} C_VEL
LIN {X 0,Y 234.109,Z 721.953,A -85,B 0,C 180,E1 -19776.562,E2 -19776.562} C_VEL
LIN {X 0,Y 233.426,Z 729.335,A -85,B 0,C 180,E1 -19779.342,E2 -19779.342} C_VEL
LIN {X 0,Y 232.976,Z 735.283,A -85,B 0,C 180,E1 -19782.252,E2 -19782.252} C_VEL
LIN {X 0,Y 232.794,Z 739.578,A -85,B 0,C 180,E1 -19785.041,E2 -19785.041} C_VEL
LIN {X 0,Y 232.824,Z 742.621,A -85,B 0,C 180,E1 -19787.802,E2 -19787.802} C_VEL
LIN {X 0,Y 232.984,Z 743.885,A -85,B 0,C 180,E1 -19789.444,E2 -19789.444} C_VEL
LIN {X 0,Y 232.571,Z 744.838,A -85,B 0,C 180,E1 -19790.876,E2 -19790.876} C_VEL
LIN {X 0,Y 230.281,Z 745.762,A -85,B 0,C 180,E1 -19793.256,E2 -19793.256} C_VEL
LIN {X 0,Y 228.517,Z 745.918,A -85,B 0,C 180,E1 -19795.201,E2 -19795.201} C_VEL
LIN {X 0,Y 228.183,Z 745.693,A -85,B 0,C 180,E1 -19796.936,E2 -19796.936} C_VEL
LIN {X 0,Y 228.287,Z 745.563,A -85,B 0,C 180,E1 -19797.183,E2 -19797.183} C_VEL
LIN {X 0,Y 230.012,Z 744.211,A -85,B 0,C 180,E1 -19800.001,E2 -19800.001} C_VEL
LIN {X 0,Y 232.208,Z 741.729,A -85,B 0,C 180,E1 -19802.786,E2 -19802.786} C_VEL
LIN {X 0,Y 235.419,Z 737.334,A -85,B 0,C 180,E1 -19805.998,E2 -19805.998} C_VEL
LIN {X 0,Y 238.556,Z 732.518,A -85,B 0,C 180,E1 -19808.471,E2 -19808.471} C_VEL
LIN {X 0,Y 242.645,Z 725.393,A -85,B 0,C 180,E1 -19811.275,E2 -19811.275} C_VEL
LIN {X 0,Y 246.721,Z 717.614,A -85,B 0,C 180,E1 -19813.603,E2 -19813.603} C_VEL
LIN {X 0,Y 251.02,Z 708.092,A -85,B 0,C 180,E1 -19815.842,E2 -19815.842} C_VEL
LIN {X 0,Y 254.963,Z 698.393,A -85,B 0,C 180,E1 -19817.651,E2 -19817.651} C_VEL
LIN {X 0,Y 259.186,Z 686.239,A -85,B 0,C 180,E1 -19819.401,E2 -19819.401} C_VEL
LIN {X 0,Y 262.845,Z 673.633,A -85,B 0,C 180,E1 -19820.791,E2 -19820.791} C_VEL
LIN {X 0,Y 265.82,Z 660.885,A -85,B 0,C 180,E1 -19821.882,E2 -19821.882} C_VEL
LIN {X 0,Y 268.222,Z 647.107,A -85,B 0,C 180,E1 -19822.723,E2 -19822.723} C_VEL
LIN {X 0,Y 277.921,Z 578.513,A -85,B 0,C 180,E1 -19825.59,E2 -19825.59} C_VEL
LIN {X 0,Y 275.953,Z 572.867,A -85,B 0,C 180,E1 -19827.168,E2 -19827.168} C_VEL
LIN {X 0,Y 273.595,Z 566.896,A -85,B 0,C 180,E1 -19829.363,E2 -19829.363} C_VEL
LIN {X 0,Y 271.751,Z 562.701,A -85,B 0,C 180,E1 -19831.514,E2 -19831.514} C_VEL
LIN {X 0,Y 270.237,Z 559.531,A -85,B 0,C 180,E1 -19834.064,E2 -19834.064} C_VEL
LIN {X 0,Y 269.517,Z 557.842,A -85,B 0,C 180,E1 -19836.459,E2 -19836.459} C_VEL
LIN {X 0,Y 269.465,Z 557.319,A -85,B 0,C 180,E1 -19838.753,E2 -19838.753} C_VEL
LIN {X 0,Y 270.208,Z 557.818,A -85,B 0,C 180,E1 -19841.335,E2 -19841.335} C_VEL
LIN {X 0,Y 271.598,Z 559.473,A -85,B 0,C 180,E1 -19843.707,E2 -19843.707} C_VEL
LIN {X 0,Y 272.729,Z 561.132,A -85,B 0,C 180,E1 -19845.155,E2 -19845.155} C_VEL
LIN {X 0,Y 273.936,Z 567.695,A -85,B 0,C 180,E1 -19847.109,E2 -19847.109} C_VEL
LIN {X 0,Y 274.832,Z 572.546,A -85,B 0,C 180,E1 -19848.297,E2 -19848.297} C_VEL
LIN {X 0,Y 274.478,Z 586.611,A -85,B 0,C 180,E1 -19849.856,E2 -19849.856} C_VEL
LIN {X 0,Y 273.952,Z 601.035,A -85,B 0,C 180,E1 -19851.166,E2 -19851.166} C_VEL
LIN {X 0,Y 272.808,Z 615.776,A -85,B 0,C 180,E1 -19852.201,E2 -19852.201} C_VEL
LIN {X 0,Y 265.824,Z 665.569,A -85,B 0,C 180,E1 -19854.314,E2 -19854.314} C_VEL
LIN {X 0,Y 262.851,Z 679.625,A -85,B 0,C 180,E1 -19855.141,E2 -19855.141} C_VEL
LIN {X 0,Y 259.316,Z 692.94,A -85,B 0,C 180,E1 -19856.246,E2 -19856.246} C_VEL
LIN {X 0,Y 255.346,Z 705.115,A -85,B 0,C 180,E1 -19857.537,E2 -19857.537} C_VEL
LIN {X 0,Y 250.871,Z 717.18,A -85,B 0,C 180,E1 -19859.249,E2 -19859.249} C_VEL
LIN {X 0,Y 245.997,Z 728.831,A -85,B 0,C 180,E1 -19861.407,E2 -19861.407} C_VEL
LIN {X 0,Y 241.565,Z 738.362,A -85,B 0,C 180,E1 -19863.658,E2 -19863.658} C_VEL
LIN {X 0,Y 237.702,Z 746.074,A -85,B 0,C 180,E1 -19866.01,E2 -19866.01} C_VEL
LIN {X 0,Y 233.849,Z 753.414,A -85,B 0,C 180,E1 -19868.857,E2 -19868.857} C_VEL
LIN {X 0,Y 231.371,Z 758.366,A -85,B 0,C 180,E1 -19871.398,E2 -19871.398} C_VEL
LIN {X 0,Y 229.213,Z 762.253,A -85,B 0,C 180,E1 -19873.978,E2 -19873.978} C_VEL
LIN {X 0,Y 228.012,Z 764.334,A -85,B 0,C 180,E1 -19875.722,E2 -19875.722} C_VEL
LIN {X 0,Y 226.578,Z 767.171,A -85,B 0,C 180,E1 -19879.271,E2 -19879.271} C_VEL
LIN {X 0,Y 225.905,Z 768.437,A -85,B 0,C 180,E1 -19882.849,E2 -19882.849} C_VEL
LIN {X 0,Y 225.886,Z 768.427,A -85,B 0,C 180,E1 -19884.641,E2 -19884.641} C_VEL
LIN {X 0,Y 225.98,Z 768.008,A -85,B 0,C 180,E1 -19886.431,E2 -19886.431} C_VEL
LIN {X 0,Y 226.09,Z 767.173,A -85,B 0,C 180,E1 -19888.216,E2 -19888.216} C_VEL
LIN {X 0,Y 226.487,Z 765.925,A -85,B 0,C 180,E1 -19889.997,E2 -19889.997} C_VEL
LIN {X 0,Y 226.294,Z 763.034,A -85,B 0,C 180,E1 -19892.667,E2 -19892.667} C_VEL
LIN {X 0,Y 226.35,Z 758.078,A -85,B 0,C 180,E1 -19895.821,E2 -19895.821} C_VEL
LIN {X 0,Y 226.481,Z 751.402,A -85,B 0,C 180,E1 -19898.923,E2 -19898.923} C_VEL
LIN {X 0,Y 226.866,Z 743.872,A -85,B 0,C 180,E1 -19901.613,E2 -19901.613} C_VEL
LIN {X 0,Y 227.571,Z 736.173,A -85,B 0,C 180,E1 -19903.844,E2 -19903.844} C_VEL
LIN {X 0,Y 228.526,Z 726.788,A -85,B 0,C 180,E1 -19906.065,E2 -19906.065} C_VEL
LIN {X 0,Y 229.768,Z 715.879,A -85,B 0,C 180,E1 -19908.135,E2 -19908.135} C_VEL
LIN {X 0,Y 230.842,Z 706.884,A -85,B 0,C 180,E1 -19909.563,E2 -19909.563} C_VEL
LIN {X 0,Y 232.445,Z 696.024,A -85,B 0,C 180,E1 -19911.736,E2 -19911.736} C_VEL
LIN {X 0,Y 234.293,Z 685.37,A -85,B 0,C 180,E1 -19913.416,E2 -19913.416} C_VEL
LIN {X 0,Y 236.072,Z 673.569,A -85,B 0,C 180,E1 -19914.863,E2 -19914.863} C_VEL
LIN {X 0,Y 237.571,Z 661.293,A -85,B 0,C 180,E1 -19915.985,E2 -19915.985} C_VEL
LIN {X 0,Y 238.717,Z 648.145,A -85,B 0,C 180,E1 -19916.835,E2 -19916.835} C_VEL
LIN {X 0,Y 239.409,Z 633.828,A -85,B 0,C 180,E1 -19917.384,E2 -19917.384} C_VEL
LIN {X 0,Y 240.002,Z 606.653,A -85,B 0,C 180,E1 -19918.197,E2 -19918.197} C_VEL
LIN {X 0,Y 235.017,Z 543.297,A -85,B 0,C 180,E1 -19920.779,E2 -19920.779} C_VEL
LIN {X 0,Y 233.904,Z 531.453,A -85,B 0,C 180,E1 -19921.34,E2 -19921.34} C_VEL
LIN {X 0,Y 234.587,Z 526.669,A -85,B 0,C 180,E1 -19922.63,E2 -19922.63} C_VEL
LIN {X 0,Y 232.518,Z 515.986,A -85,B 0,C 180,E1 -19926.005,E2 -19926.005} C_VEL
LIN {X 0,Y 230.165,Z 505.429,A -85,B 0,C 180,E1 -19929.557,E2 -19929.557} C_VEL
LIN {X 0,Y 227.834,Z 496.198,A -85,B 0,C 180,E1 -19932.955,E2 -19932.955} C_VEL
LIN {X 0,Y 227.797,Z 496.108,A -85,B 0,C 180,E1 -19937.254,E2 -19937.254} C_VEL
LIN {X 0,Y 227.834,Z 496.104,A -85,B 0,C 180,E1 -19941.906,E2 -19941.906} C_VEL
LIN {X 0,Y 227.87,Z 496.091,A -85,B 0,C 180,E1 -19946.375,E2 -19946.375} C_VEL
LIN {X 0,Y 227.894,Z 496.087,A -85,B 0,C 180,E1 -19950.434,E2 -19950.434} C_VEL
LIN {X 0,Y 227.918,Z 496.088,A -85,B 0,C 180,E1 -19954.424,E2 -19954.424} C_VEL
LIN {X 0,Y 227.951,Z 496.083,A -85,B 0,C 180,E1 -19958.285,E2 -19958.285} C_VEL
LIN {X 0,Y 228.023,Z 496.08,A -85,B 0,C 180,E1 -19962.824,E2 -19962.824} C_VEL
LIN {X 0,Y 228.082,Z 496.063,A -85,B 0,C 180,E1 -19967.543,E2 -19967.543} C_VEL
LIN {X 0,Y 228.294,Z 496.041,A -85,B 0,C 180,E1 -19971.145,E2 -19971.145} C_VEL
LIN {X 0,Y 228.342,Z 496.041,A -85,B 0,C 180,E1 -19972.928,E2 -19972.928} C_VEL
LIN {X 0,Y 228.541,Z 495.995,A -85,B 0,C 180,E1 -19978.237,E2 -19978.237} C_VEL
LIN {X 0,Y 228.542,Z 496.01,A -85,B 0,C 180,E1 -19981.762,E2 -19981.762} C_VEL
LIN {X 0,Y 228.342,Z 496.027,A -85,B 0,C 180,E1 -19987.071,E2 -19987.071} C_VEL
LIN {X 0,Y 228.15,Z 496.05,A -85,B 0,C 180,E1 -19990.65,E2 -19990.65} C_VEL
LIN {X 0,Y 228.052,Z 496.078,A -85,B 0,C 180,E1 -19994.272,E2 -19994.272} C_VEL
LIN {X 0,Y 227.99,Z 496.07,A -85,B 0,C 180,E1 -19997.954,E2 -19997.954} C_VEL
LIN {X 0,Y 227.917,Z 496.088,A -85,B 0,C 180,E1 -20002.33,E2 -20002.33} C_VEL
LIN {X 0,Y 227.931,Z 496.085,A -85,B 0,C 180,E1 -20006.604,E2 -20006.604} C_VEL
LIN {X 0,Y 227.896,Z 496.084,A -85,B 0,C 180,E1 -20010.297,E2 -20010.297} C_VEL
LIN {X 0,Y 227.865,Z 496.099,A -85,B 0,C 180,E1 -20013.722,E2 -20013.722} C_VEL
LIN {X 0,Y 227.835,Z 496.09,A -85,B 0,C 180,E1 -20018.092,E2 -20018.092} C_VEL
LIN {X 0,Y 227.826,Z 496.103,A -85,B 0,C 180,E1 -20022.738,E2 -20022.738} C_VEL
LIN {X 0,Y 227.907,Z 496.097,A -85,B 0,C 180,E1 -20027.284,E2 -20027.284} C_VEL
LIN {X 0,Y 227.862,Z 496.073,A -85,B 0,C 180,E1 -20031.917,E2 -20031.917} C_VEL
LIN {X 0,Y 227.882,Z 496.089,A -85,B 0,C 180,E1 -20036.375,E2 -20036.375} C_VEL
LIN {X 0,Y 227.91,Z 496.081,A -85,B 0,C 180,E1 -20040.44,E2 -20040.44} C_VEL
LIN {X 0,Y 227.922,Z 496.088,A -85,B 0,C 180,E1 -20044.429,E2 -20044.429} C_VEL
LIN {X 0,Y 227.956,Z 496.072,A -85,B 0,C 180,E1 -20048.29,E2 -20048.29} C_VEL
LIN {X 0,Y 228.055,Z 496.18,A -85,B 0,C 180,E1 -20052.808,E2 -20052.808} C_VEL
LIN {X 0,Y 228.26,Z 497.048,A -85,B 0,C 180,E1 -20053.164,E2 -20053.164} C_VEL
LIN {X 0,Y 235.218,Z 511.761,A -85,B 0,C 180,E1 -20054.552,E2 -20054.552} C_VEL
LIN {X 0,Y 241.741,Z 527.181,A -85,B 0,C 180,E1 -20055.782,E2 -20055.782} C_VEL
LIN {X 0,Y 240.768,Z 579.681,A -85,B 0,C 180,E1 -20057.405,E2 -20057.405} C_VEL
LIN {X 0,Y 240.337,Z 592.693,A -85,B 0,C 180,E1 -20058.127,E2 -20058.127} C_VEL
LIN {X 0,Y 239.517,Z 605.971,A -85,B 0,C 180,E1 -20059.222,E2 -20059.222} C_VEL
LIN {X 0,Y 238.488,Z 617.111,A -85,B 0,C 180,E1 -20060.461,E2 -20060.461} C_VEL
LIN {X 0,Y 237.01,Z 628.677,A -85,B 0,C 180,E1 -20062.12,E2 -20062.12} C_VEL
LIN {X 0,Y 235.51,Z 639.073,A -85,B 0,C 180,E1 -20064.008,E2 -20064.008} C_VEL
LIN {X 0,Y 233.966,Z 648.478,A -85,B 0,C 180,E1 -20066.128,E2 -20066.128} C_VEL
LIN {X 0,Y 232.621,Z 656.189,A -85,B 0,C 180,E1 -20068.272,E2 -20068.272} C_VEL
LIN {X 0,Y 231.276,Z 663.742,A -85,B 0,C 180,E1 -20070.873,E2 -20070.873} C_VEL
LIN {X 0,Y 230.165,Z 669.846,A -85,B 0,C 180,E1 -20073.504,E2 -20073.504} C_VEL
LIN {X 0,Y 229.301,Z 674.71,A -85,B 0,C 180,E1 -20076.161,E2 -20076.161} C_VEL
LIN {X 0,Y 228.777,Z 678.456,A -85,B 0,C 180,E1 -20078.838,E2 -20078.838} C_VEL
LIN {X 0,Y 228.569,Z 680.411,A -85,B 0,C 180,E1 -20080.634,E2 -20080.634} C_VEL
LIN {X 0,Y 228.497,Z 681.896,A -85,B 0,C 180,E1 -20082.436,E2 -20082.436} C_VEL
LIN {X 0,Y 228.746,Z 683.662,A -85,B 0,C 180,E1 -20086.055,E2 -20086.055} C_VEL
LIN {X 0,Y 229.166,Z 683.928,A -85,B 0,C 180,E1 -20088.068,E2 -20088.068} C_VEL
LIN {X 0,Y 230.252,Z 683.218,A -85,B 0,C 180,E1 -20091.489,E2 -20091.489} C_VEL
LIN {X 0,Y 231.779,Z 681.304,A -85,B 0,C 180,E1 -20094.543,E2 -20094.543} C_VEL
LIN {X 0,Y 233.823,Z 677.835,A -85,B 0,C 180,E1 -20097.77,E2 -20097.77} C_VEL
LIN {X 0,Y 235.984,Z 673.716,A -85,B 0,C 180,E1 -20100.42,E2 -20100.42} C_VEL
LIN {X 0,Y 238.462,Z 668.331,A -85,B 0,C 180,E1 -20103.044,E2 -20103.044} C_VEL
LIN {X 0,Y 241.335,Z 661.48,A -85,B 0,C 180,E1 -20105.624,E2 -20105.624} C_VEL
LIN {X 0,Y 243.989,Z 654.378,A -85,B 0,C 180,E1 -20107.744,E2 -20107.744} C_VEL
LIN {X 0,Y 247.093,Z 644.686,A -85,B 0,C 180,E1 -20110.045,E2 -20110.045} C_VEL
LIN {X 0,Y 249.865,Z 634.683,A -85,B 0,C 180,E1 -20111.918,E2 -20111.918} C_VEL
LIN {X 0,Y 252.246,Z 624.751,A -85,B 0,C 180,E1 -20113.39,E2 -20113.39} C_VEL
LIN {X 0,Y 254.44,Z 612.86,A -85,B 0,C 180,E1 -20114.78,E2 -20114.78} C_VEL
LIN {X 0,Y 256,Z 600.556,A -85,B 0,C 180,E1 -20115.885,E2 -20115.885} C_VEL
LIN {X 0,Y 257.046,Z 587.568,A -85,B 0,C 180,E1 -20116.716,E2 -20116.716} C_VEL
LIN {X 0,Y 257.477,Z 573.873,A -85,B 0,C 180,E1 -20117.266,E2 -20117.266} C_VEL
LIN {X 0,Y 258.059,Z 554.198,A -85,B 0,C 180,E1 -20117.865,E2 -20117.865} C_VEL
LIN {X 0,Y 257.119,Z 555.011,A -85,B 0,C 180,E1 -20118.011,E2 -20118.011} C_VEL
LIN {X 0,Y 254.538,Z 560.307,A -85,B 0,C 180,E1 -20118.309,E2 -20118.309} C_VEL
LIN {X 0,Y 251.886,Z 563.558,A -85,B 0,C 180,E1 -20118.706,E2 -20118.706} C_VEL
LIN {X 0,Y 249.246,Z 565.243,A -85,B 0,C 180,E1 -20119.17,E2 -20119.17} C_VEL
LIN {X 0,Y 248.545,Z 565.627,A -85,B 0,C 180,E1 -20119.298,E2 -20119.298} C_VEL
LIN {X 0,Y 243.915,Z 579.4,A -85,B 0,C 180,E1 -20119.726,E2 -20119.726} C_VEL
LIN {X 0,Y 241.664,Z 583.594,A -85,B 0,C 180,E1 -20120.01,E2 -20120.01} C_VEL
LIN {X 0,Y 239.984,Z 585.379,A -85,B 0,C 180,E1 -20120.289,E2 -20120.289} C_VEL
LIN {X 0,Y 238.16,Z 585.546,A -85,B 0,C 180,E1 -20120.761,E2 -20120.761} C_VEL
LIN {X 0,Y 237.415,Z 587.516,A -85,B 0,C 180,E1 -20121.15,E2 -20121.15} C_VEL
LIN {X 0,Y 236.974,Z 592.16,A -85,B 0,C 180,E1 -20121.548,E2 -20121.548} C_VEL
LIN {X 0,Y 234.609,Z 643.109,A -85,B 0,C 180,E1 -20123.827,E2 -20123.827} C_VEL
LIN {X 0,Y 233.699,Z 656.677,A -85,B 0,C 180,E1 -20124.784,E2 -20124.784} C_VEL
LIN {X 0,Y 232.709,Z 669.55,A -85,B 0,C 180,E1 -20126.034,E2 -20126.034} C_VEL
LIN {X 0,Y 231.447,Z 681.793,A -85,B 0,C 180,E1 -20127.592,E2 -20127.592} C_VEL
LIN {X 0,Y 230.157,Z 693.615,A -85,B 0,C 180,E1 -20129.493,E2 -20129.493} C_VEL
LIN {X 0,Y 228.855,Z 705.074,A -85,B 0,C 180,E1 -20131.826,E2 -20131.826} C_VEL
LIN {X 0,Y 227.975,Z 713.167,A -85,B 0,C 180,E1 -20133.842,E2 -20133.842} C_VEL
LIN {X 0,Y 227.093,Z 721.22,A -85,B 0,C 180,E1 -20136.277,E2 -20136.277} C_VEL
LIN {X 0,Y 226.347,Z 729.159,A -85,B 0,C 180,E1 -20139.301,E2 -20139.301} C_VEL
LIN {X 0,Y 225.936,Z 734.5,A -85,B 0,C 180,E1 -20141.878,E2 -20141.878} C_VEL
LIN {X 0,Y 225.695,Z 739.265,A -85,B 0,C 180,E1 -20144.876,E2 -20144.876} C_VEL
LIN {X 0,Y 225.706,Z 742.252,A -85,B 0,C 180,E1 -20147.411,E2 -20147.411} C_VEL
LIN {X 0,Y 225.897,Z 743.994,A -85,B 0,C 180,E1 -20149.502,E2 -20149.502} C_VEL
LIN {X 0,Y 226.2,Z 744.979,A -85,B 0,C 180,E1 -20151.064,E2 -20151.064} C_VEL
LIN {X 0,Y 226.655,Z 745.677,A -85,B 0,C 180,E1 -20152.876,E2 -20152.876} C_VEL
LIN {X 0,Y 227.233,Z 745.93,A -85,B 0,C 180,E1 -20154.677,E2 -20154.677} C_VEL
LIN {X 0,Y 228.287,Z 745.563,A -85,B 0,C 180,E1 -20157.183,E2 -20157.183} C_VEL
LIN {X 0,Y 228.457,Z 745.112,A -85,B 0,C 180,E1 -20158.661,E2 -20158.661} C_VEL
LIN {X 0,Y 227.277,Z 744.065,A -85,B 0,C 180,E1 -20161.125,E2 -20161.125} C_VEL
LIN {X 0,Y 226.452,Z 742.373,A -85,B 0,C 180,E1 -20163.581,E2 -20163.581} C_VEL
LIN {X 0,Y 227.161,Z 740.851,A -85,B 0,C 180,E1 -20165.01,E2 -20165.01} C_VEL
LIN {X 0,Y 230.503,Z 736.519,A -85,B 0,C 180,E1 -20167.887,E2 -20167.887} C_VEL
LIN {X 0,Y 234.013,Z 731.408,A -85,B 0,C 180,E1 -20170.382,E2 -20170.382} C_VEL
LIN {X 0,Y 237.774,Z 725.222,A -85,B 0,C 180,E1 -20172.726,E2 -20172.726} C_VEL
LIN {X 0,Y 242.244,Z 717.117,A -85,B 0,C 180,E1 -20175.136,E2 -20175.136} C_VEL
LIN {X 0,Y 246.971,Z 707.361,A -85,B 0,C 180,E1 -20177.386,E2 -20177.386} C_VEL
LIN {X 0,Y 251.64,Z 696.18,A -85,B 0,C 180,E1 -20179.37,E2 -20179.37} C_VEL
LIN {X 0,Y 255.254,Z 686.312,A -85,B 0,C 180,E1 -20180.763,E2 -20180.763} C_VEL
LIN {X 0,Y 258.946,Z 674.247,A -85,B 0,C 180,E1 -20182.096,E2 -20182.096} C_VEL
LIN {X 0,Y 262.106,Z 661.249,A -85,B 0,C 180,E1 -20183.202,E2 -20183.202} C_VEL
LIN {X 0,Y 264.799,Z 646.738,A -85,B 0,C 180,E1 -20184.084,E2 -20184.084} C_VEL
LIN {X 0,Y 274.503,Z 582.155,A -85,B 0,C 180,E1 -20186.781,E2 -20186.781} C_VEL
LIN {X 0,Y 272.727,Z 576.826,A -85,B 0,C 180,E1 -20188.447,E2 -20188.447} C_VEL
LIN {X 0,Y 271.078,Z 572.398,A -85,B 0,C 180,E1 -20190.267,E2 -20190.267} C_VEL
LIN {X 0,Y 269.752,Z 569.07,A -85,B 0,C 180,E1 -20192.075,E2 -20192.075} C_VEL
LIN {X 0,Y 268.569,Z 566.342,A -85,B 0,C 180,E1 -20194.304,E2 -20194.304} C_VEL
LIN {X 0,Y 267.92,Z 564.633,A -85,B 0,C 180,E1 -20196.869,E2 -20196.869} C_VEL
LIN {X 0,Y 267.964,Z 564.254,A -85,B 0,C 180,E1 -20199.011,E2 -20199.011} C_VEL
LIN {X 0,Y 268.625,Z 564.711,A -85,B 0,C 180,E1 -20201.26,E2 -20201.26} C_VEL
LIN {X 0,Y 270.104,Z 566.559,A -85,B 0,C 180,E1 -20203.814,E2 -20203.814} C_VEL
LIN {X 0,Y 270.699,Z 567.536,A -85,B 0,C 180,E1 -20204.627,E2 -20204.627} C_VEL
LIN {X 0,Y 271.595,Z 573.653,A -85,B 0,C 180,E1 -20206.432,E2 -20206.432} C_VEL
LIN {X 0,Y 272.013,Z 576.936,A -85,B 0,C 180,E1 -20207.242,E2 -20207.242} C_VEL
LIN {X 0,Y 271.518,Z 588.994,A -85,B 0,C 180,E1 -20208.596,E2 -20208.596} C_VEL
LIN {X 0,Y 270.642,Z 603.243,A -85,B 0,C 180,E1 -20209.929,E2 -20209.929} C_VEL
LIN {X 0,Y 269.362,Z 617.675,A -85,B 0,C 180,E1 -20210.932,E2 -20210.932} C_VEL
LIN {X 0,Y 262.211,Z 665.034,A -85,B 0,C 180,E1 -20212.968,E2 -20212.968} C_VEL
LIN {X 0,Y 259.231,Z 678.571,A -85,B 0,C 180,E1 -20213.744,E2 -20213.744} C_VEL
LIN {X 0,Y 255.762,Z 691.057,A -85,B 0,C 180,E1 -20214.754,E2 -20214.754} C_VEL
LIN {X 0,Y 251.58,Z 703.348,A -85,B 0,C 180,E1 -20216.031,E2 -20216.031} C_VEL
LIN {X 0,Y 246.797,Z 715.565,A -85,B 0,C 180,E1 -20217.725,E2 -20217.725} C_VEL
LIN {X 0,Y 242.433,Z 725.637,A -85,B 0,C 180,E1 -20219.512,E2 -20219.512} C_VEL
LIN {X 0,Y 237.563,Z 735.503,A -85,B 0,C 180,E1 -20221.746,E2 -20221.746} C_VEL
LIN {X 0,Y 233.271,Z 743.658,A -85,B 0,C 180,E1 -20224.094,E2 -20224.094} C_VEL
LIN {X 0,Y 229.601,Z 750.351,A -85,B 0,C 180,E1 -20226.548,E2 -20226.548} C_VEL
LIN {X 0,Y 226.371,Z 755.78,A -85,B 0,C 180,E1 -20229.079,E2 -20229.079} C_VEL
LIN {X 0,Y 223.889,Z 760.137,A -85,B 0,C 180,E1 -20231.702,E2 -20231.702} C_VEL
LIN {X 0,Y 222.39,Z 762.464,A -85,B 0,C 180,E1 -20233.473,E2 -20233.473} C_VEL
LIN {X 0,Y 221.119,Z 764.358,A -85,B 0,C 180,E1 -20235.267,E2 -20235.267} C_VEL
LIN {X 0,Y 219.588,Z 766.982,A -85,B 0,C 180,E1 -20238.926,E2 -20238.926} C_VEL
LIN {X 0,Y 219.091,Z 767.671,A -85,B 0,C 180,E1 -20240.767,E2 -20240.767} C_VEL
LIN {X 0,Y 218.805,Z 767.853,A -85,B 0,C 180,E1 -20244.467,E2 -20244.467} C_VEL
LIN {X 0,Y 218.912,Z 767.355,A -85,B 0,C 180,E1 -20246.316,E2 -20246.316} C_VEL
LIN {X 0,Y 219.044,Z 766.394,A -85,B 0,C 180,E1 -20248.158,E2 -20248.158} C_VEL
LIN {X 0,Y 219.446,Z 764.998,A -85,B 0,C 180,E1 -20249.997,E2 -20249.997} C_VEL
LIN {X 0,Y 219.257,Z 761.909,A -85,B 0,C 180,E1 -20252.753,E2 -20252.753} C_VEL
LIN {X 0,Y 219.293,Z 757.637,A -85,B 0,C 180,E1 -20255.514,E2 -20255.514} C_VEL
LIN {X 0,Y 219.386,Z 752.011,A -85,B 0,C 180,E1 -20258.285,E2 -20258.285} C_VEL
LIN {X 0,Y 219.695,Z 744.818,A -85,B 0,C 180,E1 -20261.063,E2 -20261.063} C_VEL
LIN {X 0,Y 220.344,Z 737.408,A -85,B 0,C 180,E1 -20263.367,E2 -20263.367} C_VEL
LIN {X 0,Y 221.389,Z 727.395,A -85,B 0,C 180,E1 -20265.887,E2 -20265.887} C_VEL
LIN {X 0,Y 222.519,Z 717.248,A -85,B 0,C 180,E1 -20267.932,E2 -20267.932} C_VEL
LIN {X 0,Y 223.677,Z 707.704,A -85,B 0,C 180,E1 -20269.579,E2 -20269.579} C_VEL
LIN {X 0,Y 225.197,Z 697.736,A -85,B 0,C 180,E1 -20271.749,E2 -20271.749} C_VEL
LIN {X 0,Y 226.965,Z 687.648,A -85,B 0,C 180,E1 -20273.492,E2 -20273.492} C_VEL
LIN {X 0,Y 228.535,Z 678.49,A -85,B 0,C 180,E1 -20274.768,E2 -20274.768} C_VEL
LIN {X 0,Y 230.33,Z 665.81,A -85,B 0,C 180,E1 -20276.134,E2 -20276.134} C_VEL
LIN {X 0,Y 231.702,Z 652.739,A -85,B 0,C 180,E1 -20277.155,E2 -20277.155} C_VEL
LIN {X 0,Y 232.596,Z 640.136,A -85,B 0,C 180,E1 -20277.798,E2 -20277.798} C_VEL
LIN {X 0,Y 233.436,Z 607.291,A -85,B 0,C 180,E1 -20278.827,E2 -20278.827} C_VEL
LIN {X 0,Y 228.633,Z 544.582,A -85,B 0,C 180,E1 -20281.461,E2 -20281.461} C_VEL
LIN {X 0,Y 227.328,Z 530.352,A -85,B 0,C 180,E1 -20282.159,E2 -20282.159} C_VEL
LIN {X 0,Y 227.514,Z 526.968,A -85,B 0,C 180,E1 -20283.126,E2 -20283.126} C_VEL
LIN {X 0,Y 225.137,Z 515.286,A -85,B 0,C 180,E1 -20286.993,E2 -20286.993} C_VEL
LIN {X 0,Y 223.011,Z 505.905,A -85,B 0,C 180,E1 -20290.292,E2 -20290.292} C_VEL
LIN {X 0,Y 220.791,Z 497.074,A -85,B 0,C 180,E1 -20293.672,E2 -20293.672} C_VEL
LIN {X 0,Y 220.759,Z 496.989,A -85,B 0,C 180,E1 -20298.044,E2 -20298.044} C_VEL
LIN {X 0,Y 220.798,Z 496.974,A -85,B 0,C 180,E1 -20300.46,E2 -20300.46} C_VEL
LIN {X 0,Y 220.792,Z 496.967,A -85,B 0,C 180,E1 -20305.043,E2 -20305.043} C_VEL
LIN {X 0,Y 220.824,Z 496.976,A -85,B 0,C 180,E1 -20309.387,E2 -20309.387} C_VEL
LIN {X 0,Y 220.884,Z 496.959,A -85,B 0,C 180,E1 -20313.547,E2 -20313.547} C_VEL
LIN {X 0,Y 220.867,Z 496.97,A -85,B 0,C 180,E1 -20317.552,E2 -20317.552} C_VEL
LIN {X 0,Y 220.973,Z 496.954,A -85,B 0,C 180,E1 -20322.57,E2 -20322.57} C_VEL
LIN {X 0,Y 221.014,Z 496.944,A -85,B 0,C 180,E1 -20327.138,E2 -20327.138} C_VEL
LIN {X 0,Y 221.224,Z 496.917,A -85,B 0,C 180,E1 -20330.86,E2 -20330.86} C_VEL
LIN {X 0,Y 221.293,Z 496.919,A -85,B 0,C 180,E1 -20332.701,E2 -20332.701} C_VEL
LIN {X 0,Y 221.499,Z 496.871,A -85,B 0,C 180,E1 -20338.181,E2 -20338.181} C_VEL
LIN {X 0,Y 221.5,Z 496.887,A -85,B 0,C 180,E1 -20341.818,E2 -20341.818} C_VEL
LIN {X 0,Y 221.277,Z 496.906,A -85,B 0,C 180,E1 -20347.298,E2 -20347.298} C_VEL
LIN {X 0,Y 221.099,Z 496.93,A -85,B 0,C 180,E1 -20350.994,E2 -20350.994} C_VEL
LIN {X 0,Y 221.004,Z 496.948,A -85,B 0,C 180,E1 -20356.63,E2 -20356.63} C_VEL
LIN {X 0,Y 220.88,Z 496.951,A -85,B 0,C 180,E1 -20360.487,E2 -20360.487} C_VEL
LIN {X 0,Y 220.855,Z 496.974,A -85,B 0,C 180,E1 -20364.436,E2 -20364.436} C_VEL
LIN {X 0,Y 220.824,Z 496.958,A -85,B 0,C 180,E1 -20368.514,E2 -20368.514} C_VEL
LIN {X 0,Y 220.806,Z 496.98,A -85,B 0,C 180,E1 -20372.757,E2 -20372.757} C_VEL
LIN {X 0,Y 220.799,Z 496.964,A -85,B 0,C 180,E1 -20377.28,E2 -20377.28} C_VEL
LIN {X 0,Y 220.775,Z 496.983,A -85,B 0,C 180,E1 -20381.95,E2 -20381.95} C_VEL
LIN {X 0,Y 220.863,Z 496.972,A -85,B 0,C 180,E1 -20387.043,E2 -20387.043} C_VEL
LIN {X 0,Y 220.849,Z 496.961,A -85,B 0,C 180,E1 -20390.476,E2 -20390.476} C_VEL
LIN {X 0,Y 220.807,Z 496.947,A -85,B 0,C 180,E1 -20395.05,E2 -20395.05} C_VEL
LIN {X 0,Y 220.86,Z 496.97,A -85,B 0,C 180,E1 -20399.398,E2 -20399.398} C_VEL
LIN {X 0,Y 220.888,Z 496.949,A -85,B 0,C 180,E1 -20403.552,E2 -20403.552} C_VEL
LIN {X 0,Y 220.872,Z 496.957,A -85,B 0,C 180,E1 -20407.556,E2 -20407.556} C_VEL
LIN {X 0,Y 220.973,Z 497.105,A -85,B 0,C 180,E1 -20411.963,E2 -20411.963} C_VEL
LIN {X 0,Y 221.169,Z 497.979,A -85,B 0,C 180,E1 -20412.283,E2 -20412.283} C_VEL
LIN {X 0,Y 227.841,Z 511.689,A -85,B 0,C 180,E1 -20413.666,E2 -20413.666} C_VEL
LIN {X 0,Y 235.285,Z 529.117,A -85,B 0,C 180,E1 -20415.14,E2 -20415.14} C_VEL
LIN {X 0,Y 234.387,Z 569.877,A -85,B 0,C 180,E1 -20416.398,E2 -20416.398} C_VEL
LIN {X 0,Y 234.173,Z 585.328,A -85,B 0,C 180,E1 -20417.007,E2 -20417.007} C_VEL
LIN {X 0,Y 233.5,Z 598.107,A -85,B 0,C 180,E1 -20417.84,E2 -20417.84} C_VEL
LIN {X 0,Y 232.674,Z 609.477,A -85,B 0,C 180,E1 -20418.901,E2 -20418.901} C_VEL
LIN {X 0,Y 231.387,Z 621.607,A -85,B 0,C 180,E1 -20420.387,E2 -20420.387} C_VEL
LIN {X 0,Y 229.864,Z 632.512,A -85,B 0,C 180,E1 -20422.095,E2 -20422.095} C_VEL
LIN {X 0,Y 228.507,Z 641.361,A -85,B 0,C 180,E1 -20423.823,E2 -20423.823} C_VEL
LIN {X 0,Y 226.942,Z 650.473,A -85,B 0,C 180,E1 -20426.007,E2 -20426.007} C_VEL
LIN {X 0,Y 225.241,Z 659.663,A -85,B 0,C 180,E1 -20428.759,E2 -20428.759} C_VEL
LIN {X 0,Y 223.968,Z 666.543,A -85,B 0,C 180,E1 -20431.352,E2 -20431.352} C_VEL
LIN {X 0,Y 223.04,Z 671.407,A -85,B 0,C 180,E1 -20433.616,E2 -20433.616} C_VEL
LIN {X 0,Y 222.204,Z 676.15,A -85,B 0,C 180,E1 -20436.359,E2 -20436.359} C_VEL
LIN {X 0,Y 221.706,Z 679.786,A -85,B 0,C 180,E1 -20439.123,E2 -20439.123} C_VEL
LIN {X 0,Y 221.512,Z 681.654,A -85,B 0,C 180,E1 -20440.977,E2 -20440.977} C_VEL
LIN {X 0,Y 221.462,Z 683.075,A -85,B 0,C 180,E1 -20442.838,E2 -20442.838} C_VEL
LIN {X 0,Y 221.547,Z 684.105,A -85,B 0,C 180,E1 -20444.704,E2 -20444.704} C_VEL
LIN {X 0,Y 221.802,Z 684.737,A -85,B 0,C 180,E1 -20446.572,E2 -20446.572} C_VEL
LIN {X 0,Y 222.227,Z 684.918,A -85,B 0,C 180,E1 -20448.439,E2 -20448.439} C_VEL
LIN {X 0,Y 222.787,Z 684.706,A -85,B 0,C 180,E1 -20450.307,E2 -20450.307} C_VEL
LIN {X 0,Y 223.498,Z 684.102,A -85,B 0,C 180,E1 -20452.172,E2 -20452.172} C_VEL
LIN {X 0,Y 225.032,Z 682.258,A -85,B 0,C 180,E1 -20455.084,E2 -20455.084} C_VEL
LIN {X 0,Y 227.391,Z 678.453,A -85,B 0,C 180,E1 -20458.627,E2 -20458.627} C_VEL
LIN {X 0,Y 229.707,Z 674.216,A -85,B 0,C 180,E1 -20461.344,E2 -20461.344} C_VEL
LIN {X 0,Y 232.35,Z 668.704,A -85,B 0,C 180,E1 -20464.03,E2 -20464.03} C_VEL
LIN {X 0,Y 235.376,Z 661.68,A -85,B 0,C 180,E1 -20466.671,E2 -20466.671} C_VEL
LIN {X 0,Y 238.806,Z 652.721,A -85,B 0,C 180,E1 -20469.256,E2 -20469.256} C_VEL
LIN {X 0,Y 241.899,Z 643.16,A -85,B 0,C 180,E1 -20471.439,E2 -20471.439} C_VEL
LIN {X 0,Y 244.759,Z 632.811,A -85,B 0,C 180,E1 -20473.282,E2 -20473.282} C_VEL
LIN {X 0,Y 247.491,Z 621.03,A -85,B 0,C 180,E1 -20474.919,E2 -20474.919} C_VEL
LIN {X 0,Y 249.499,Z 609.067,A -85,B 0,C 180,E1 -20476.208,E2 -20476.208} C_VEL
LIN {X 0,Y 250.954,Z 596.365,A -85,B 0,C 180,E1 -20477.227,E2 -20477.227} C_VEL
LIN {X 0,Y 251.769,Z 583.664,A -85,B 0,C 180,E1 -20477.938,E2 -20477.938} C_VEL
LIN {X 0,Y 252.058,Z 572.668,A -85,B 0,C 180,E1 -20478.332,E2 -20478.332} C_VEL
LIN {X 0,Y 247.713,Z 583.922,A -85,B 0,C 180,E1 -20478.729,E2 -20478.729} C_VEL
LIN {X 0,Y 245.141,Z 588.131,A -85,B 0,C 180,E1 -20479.02,E2 -20479.02} C_VEL
LIN {X 0,Y 242.385,Z 591.056,A -85,B 0,C 180,E1 -20479.415,E2 -20479.415} C_VEL
LIN {X 0,Y 239.551,Z 592.594,A -85,B 0,C 180,E1 -20479.926,E2 -20479.926} C_VEL
LIN {X 0,Y 236.147,Z 599.32,A -85,B 0,C 180,E1 -20480.125,E2 -20480.125} C_VEL
LIN {X 0,Y 234.058,Z 602.036,A -85,B 0,C 180,E1 -20480.352,E2 -20480.352} C_VEL
LIN {X 0,Y 232.495,Z 603.271,A -85,B 0,C 180,E1 -20480.596,E2 -20480.596} C_VEL
LIN {X 0,Y 231.165,Z 603.59,A -85,B 0,C 180,E1 -20480.888,E2 -20480.888} C_VEL
LIN {X 0,Y 230.368,Z 603.365,A -85,B 0,C 180,E1 -20481.149,E2 -20481.149} C_VEL
LIN {X 0,Y 229.637,Z 604.962,A -85,B 0,C 180,E1 -20481.563,E2 -20481.563} C_VEL
LIN {X 0,Y 229.253,Z 608.647,A -85,B 0,C 180,E1 -20481.907,E2 -20481.907} C_VEL
LIN {X 0,Y 227.558,Z 644.388,A -85,B 0,C 180,E1 -20483.601,E2 -20483.601} C_VEL
LIN {X 0,Y 226.565,Z 659.03,A -85,B 0,C 180,E1 -20484.709,E2 -20484.709} C_VEL
LIN {X 0,Y 225.4,Z 672.464,A -85,B 0,C 180,E1 -20486.129,E2 -20486.129} C_VEL
LIN {X 0,Y 224.099,Z 685.072,A -85,B 0,C 180,E1 -20487.865,E2 -20487.865} C_VEL
LIN {X 0,Y 222.716,Z 696.787,A -85,B 0,C 180,E1 -20489.938,E2 -20489.938} C_VEL
LIN {X 0,Y 221.63,Z 706.244,A -85,B 0,C 180,E1 -20491.996,E2 -20491.996} C_VEL
LIN {X 0,Y 220.585,Z 715.681,A -85,B 0,C 180,E1 -20494.526,E2 -20494.526} C_VEL
LIN {X 0,Y 219.685,Z 724.401,A -85,B 0,C 180,E1 -20497.426,E2 -20497.426} C_VEL
LIN {X 0,Y 219.072,Z 731.233,A -85,B 0,C 180,E1 -20500.316,E2 -20500.316} C_VEL
LIN {X 0,Y 218.732,Z 736.6,A -85,B 0,C 180,E1 -20503.192,E2 -20503.192} C_VEL
LIN {X 0,Y 218.586,Z 740.663,A -85,B 0,C 180,E1 -20506.047,E2 -20506.047} C_VEL
LIN {X 0,Y 218.712,Z 743.565,A -85,B 0,C 180,E1 -20508.884,E2 -20508.884} C_VEL
LIN {X 0,Y 219.027,Z 744.929,A -85,B 0,C 180,E1 -20510.768,E2 -20510.768} C_VEL
LIN {X 0,Y 219.557,Z 745.938,A -85,B 0,C 180,E1 -20512.91,E2 -20512.91} C_VEL
LIN {X 0,Y 220.782,Z 746.431,A -85,B 0,C 180,E1 -20516.35,E2 -20516.35} C_VEL
LIN {X 0,Y 222.863,Z 745.306,A -85,B 0,C 180,E1 -20520.001,E2 -20520.001} C_VEL
LIN {X 0,Y 225.207,Z 743.125,A -85,B 0,C 180,E1 -20522.966,E2 -20522.966} C_VEL
LIN {X 0,Y 227.161,Z 740.851,A -85,B 0,C 180,E1 -20525.01,E2 -20525.01} C_VEL
LIN {X 0,Y 228.024,Z 739.159,A -85,B 0,C 180,E1 -20526.421,E2 -20526.421} C_VEL
LIN {X 0,Y 228.101,Z 736.308,A -85,B 0,C 180,E1 -20528.811,E2 -20528.811} C_VEL
LIN {X 0,Y 228.508,Z 732.846,A -85,B 0,C 180,E1 -20531.131,E2 -20531.131} C_VEL
LIN {X 0,Y 229.838,Z 730.181,A -85,B 0,C 180,E1 -20532.4,E2 -20532.4} C_VEL
LIN {X 0,Y 234.124,Z 723.504,A -85,B 0,C 180,E1 -20534.783,E2 -20534.783} C_VEL
LIN {X 0,Y 238.856,Z 715.154,A -85,B 0,C 180,E1 -20537.112,E2 -20537.112} C_VEL
LIN {X 0,Y 243.172,Z 706.695,A -85,B 0,C 180,E1 -20538.975,E2 -20538.975} C_VEL
LIN {X 0,Y 247.332,Z 697.281,A -85,B 0,C 180,E1 -20540.653,E2 -20540.653} C_VEL
LIN {X 0,Y 251.785,Z 685.641,A -85,B 0,C 180,E1 -20542.277,E2 -20542.277} C_VEL
LIN {X 0,Y 255.946,Z 672.636,A -85,B 0,C 180,E1 -20543.678,E2 -20543.678} C_VEL
LIN {X 0,Y 259.238,Z 659.413,A -85,B 0,C 180,E1 -20544.741,E2 -20544.741} C_VEL
LIN {X 0,Y 261.693,Z 646.281,A -85,B 0,C 180,E1 -20545.502,E2 -20545.502} C_VEL
LIN {X 0,Y 271.326,Z 585.883,A -85,B 0,C 180,E1 -20548.036,E2 -20548.036} C_VEL
LIN {X 0,Y 269.703,Z 580.917,A -85,B 0,C 180,E1 -20549.829,E2 -20549.829} C_VEL
LIN {X 0,Y 268.444,Z 577.256,A -85,B 0,C 180,E1 -20551.517,E2 -20551.517} C_VEL
LIN {X 0,Y 267.298,Z 574.194,A -85,B 0,C 180,E1 -20553.515,E2 -20553.515} C_VEL
LIN {X 0,Y 266.504,Z 572.162,A -85,B 0,C 180,E1 -20555.75,E2 -20555.75} C_VEL
LIN {X 0,Y 266.316,Z 571.295,A -85,B 0,C 180,E1 -20557.653,E2 -20557.653} C_VEL
LIN {X 0,Y 266.876,Z 571.499,A -85,B 0,C 180,E1 -20560.833,E2 -20560.833} C_VEL
LIN {X 0,Y 268.063,Z 573.016,A -85,B 0,C 180,E1 -20563.195,E2 -20563.195} C_VEL
LIN {X 0,Y 268.706,Z 573.988,A -85,B 0,C 180,E1 -20564.101,E2 -20564.101} C_VEL
LIN {X 0,Y 269.391,Z 580.423,A -85,B 0,C 180,E1 -20565.965,E2 -20565.965} C_VEL
LIN {X 0,Y 269.385,Z 582.188,A -85,B 0,C 180,E1 -20566.258,E2 -20566.258} C_VEL
LIN {X 0,Y 268.582,Z 593.369,A -85,B 0,C 180,E1 -20567.506,E2 -20567.506} C_VEL
LIN {X 0,Y 267.612,Z 606.418,A -85,B 0,C 180,E1 -20568.721,E2 -20568.721} C_VEL
LIN {X 0,Y 266.181,Z 619.273,A -85,B 0,C 180,E1 -20569.609,E2 -20569.609} C_VEL
LIN {X 0,Y 258.985,Z 664.522,A -85,B 0,C 180,E1 -20571.564,E2 -20571.564} C_VEL
LIN {X 0,Y 255.523,Z 678.944,A -85,B 0,C 180,E1 -20572.389,E2 -20572.389} C_VEL
LIN {X 0,Y 251.364,Z 692.694,A -85,B 0,C 180,E1 -20573.546,E2 -20573.546} C_VEL
LIN {X 0,Y 246.492,Z 705.817,A -85,B 0,C 180,E1 -20574.981,E2 -20574.981} C_VEL
LIN {X 0,Y 242.003,Z 716.402,A -85,B 0,C 180,E1 -20576.508,E2 -20576.508} C_VEL
LIN {X 0,Y 236.531,Z 727.796,A -85,B 0,C 180,E1 -20578.666,E2 -20578.666} C_VEL
LIN {X 0,Y 231.5,Z 737.237,A -85,B 0,C 180,E1 -20580.936,E2 -20580.936} C_VEL
LIN {X 0,Y 227.022,Z 744.896,A -85,B 0,C 180,E1 -20583.325,E2 -20583.325} C_VEL
LIN {X 0,Y 222.484,Z 752.263,A -85,B 0,C 180,E1 -20586.296,E2 -20586.296} C_VEL
LIN {X 0,Y 219.762,Z 756.375,A -85,B 0,C 180,E1 -20588.419,E2 -20588.419} C_VEL
LIN {X 0,Y 216.361,Z 761.599,A -85,B 0,C 180,E1 -20592.023,E2 -20592.023} C_VEL
LIN {X 0,Y 214.249,Z 764.409,A -85,B 0,C 180,E1 -20594.783,E2 -20594.783} C_VEL
LIN {X 0,Y 213.277,Z 765.766,A -85,B 0,C 180,E1 -20596.661,E2 -20596.661} C_VEL
LIN {X 0,Y 212.063,Z 767.286,A -85,B 0,C 180,E1 -20600.459,E2 -20600.459} C_VEL
LIN {X 0,Y 211.792,Z 767.473,A -85,B 0,C 180,E1 -20602.369,E2 -20602.369} C_VEL
LIN {X 0,Y 211.751,Z 767.139,A -85,B 0,C 180,E1 -20604.689,E2 -20604.689} C_VEL
LIN {X 0,Y 212.019,Z 765.538,A -85,B 0,C 180,E1 -20608.097,E2 -20608.097} C_VEL
LIN {X 0,Y 212.404,Z 764.067,A -85,B 0,C 180,E1 -20609.997,E2 -20609.997} C_VEL
LIN {X 0,Y 212.223,Z 760.782,A -85,B 0,C 180,E1 -20612.844,E2 -20612.844} C_VEL
LIN {X 0,Y 212.244,Z 756.288,A -85,B 0,C 180,E1 -20615.698,E2 -20615.698} C_VEL
LIN {X 0,Y 212.372,Z 750.375,A -85,B 0,C 180,E1 -20618.561,E2 -20618.561} C_VEL
LIN {X 0,Y 212.724,Z 742.849,A -85,B 0,C 180,E1 -20621.43,E2 -20621.43} C_VEL
LIN {X 0,Y 213.422,Z 735.154,A -85,B 0,C 180,E1 -20623.809,E2 -20623.809} C_VEL
LIN {X 0,Y 214.399,Z 725.765,A -85,B 0,C 180,E1 -20626.175,E2 -20626.175} C_VEL
LIN {X 0,Y 215.738,Z 714.151,A -85,B 0,C 180,E1 -20628.516,E2 -20628.516} C_VEL
LIN {X 0,Y 216.377,Z 709.011,A -85,B 0,C 180,E1 -20629.464,E2 -20629.464} C_VEL
LIN {X 0,Y 217.973,Z 699.237,A -85,B 0,C 180,E1 -20631.761,E2 -20631.761} C_VEL
LIN {X 0,Y 219.943,Z 688.383,A -85,B 0,C 180,E1 -20633.788,E2 -20633.788} C_VEL
LIN {X 0,Y 221.784,Z 677.928,A -85,B 0,C 180,E1 -20635.324,E2 -20635.324} C_VEL
LIN {X 0,Y 223.641,Z 665.407,A -85,B 0,C 180,E1 -20636.726,E2 -20636.726} C_VEL
LIN {X 0,Y 225.083,Z 652.178,A -85,B 0,C 180,E1 -20637.798,E2 -20637.798} C_VEL
LIN {X 0,Y 226.046,Z 638.812,A -85,B 0,C 180,E1 -20638.499,E2 -20638.499} C_VEL
LIN {X 0,Y 226.884,Z 607.935,A -85,B 0,C 180,E1 -20639.491,E2 -20639.491} C_VEL
LIN {X 0,Y 222.27,Z 545.972,A -85,B 0,C 180,E1 -20642.179,E2 -20642.179} C_VEL
LIN {X 0,Y 220.687,Z 529.708,A -85,B 0,C 180,E1 -20642.977,E2 -20642.977} C_VEL
LIN {X 0,Y 220.196,Z 526.512,A -85,B 0,C 180,E1 -20643.916,E2 -20643.916} C_VEL
LIN {X 0,Y 217.987,Z 515.349,A -85,B 0,C 180,E1 -20647.771,E2 -20647.771} C_VEL
LIN {X 0,Y 215.253,Z 503.863,A -85,B 0,C 180,E1 -20652.03,E2 -20652.03} C_VEL
LIN {X 0,Y 213.757,Z 497.957,A -85,B 0,C 180,E1 -20654.431,E2 -20654.431} C_VEL
LIN {X 0,Y 213.708,Z 497.862,A -85,B 0,C 180,E1 -20659.14,E2 -20659.14} C_VEL
LIN {X 0,Y 213.735,Z 497.856,A -85,B 0,C 180,E1 -20663.709,E2 -20663.709} C_VEL
LIN {X 0,Y 213.771,Z 497.856,A -85,B 0,C 180,E1 -20668.729,E2 -20668.729} C_VEL
LIN {X 0,Y 213.816,Z 497.831,A -85,B 0,C 180,E1 -20672.601,E2 -20672.601} C_VEL
LIN {X 0,Y 213.841,Z 497.846,A -85,B 0,C 180,E1 -20676.951,E2 -20676.951} C_VEL
LIN {X 0,Y 213.932,Z 497.833,A -85,B 0,C 180,E1 -20682.802,E2 -20682.802} C_VEL
LIN {X 0,Y 213.969,Z 497.823,A -85,B 0,C 180,E1 -20686.707,E2 -20686.707} C_VEL
LIN {X 0,Y 214.155,Z 497.793,A -85,B 0,C 180,E1 -20690.555,E2 -20690.555} C_VEL
LIN {X 0,Y 214.228,Z 497.797,A -85,B 0,C 180,E1 -20692.459,E2 -20692.459} C_VEL
LIN {X 0,Y 214.432,Z 497.75,A -85,B 0,C 180,E1 -20698.121,E2 -20698.121} C_VEL
LIN {X 0,Y 214.537,Z 497.741,A -85,B 0,C 180,E1 -20699.999,E2 -20699.999} C_VEL
LIN {X 0,Y 214.433,Z 497.767,A -85,B 0,C 180,E1 -20701.878,E2 -20701.878} C_VEL
LIN {X 0,Y 214.215,Z 497.783,A -85,B 0,C 180,E1 -20707.54,E2 -20707.54} C_VEL
LIN {X 0,Y 214.032,Z 497.814,A -85,B 0,C 180,E1 -20711.362,E2 -20711.362} C_VEL
LIN {X 0,Y 213.921,Z 497.835,A -85,B 0,C 180,E1 -20715.237,E2 -20715.237} C_VEL
LIN {X 0,Y 213.826,Z 497.824,A -85,B 0,C 180,E1 -20719.188,E2 -20719.188} C_VEL
LIN {X 0,Y 213.835,Z 497.848,A -85,B 0,C 180,E1 -20723.228,E2 -20723.228} C_VEL
LIN {X 0,Y 213.817,Z 497.836,A -85,B 0,C 180,E1 -20727.451,E2 -20727.451} C_VEL
LIN {X 0,Y 213.765,Z 497.854,A -85,B 0,C 180,E1 -20731.737,E2 -20731.737} C_VEL
LIN {X 0,Y 213.732,Z 497.848,A -85,B 0,C 180,E1 -20736.29,E2 -20736.29} C_VEL
LIN {X 0,Y 213.712,Z 497.865,A -85,B 0,C 180,E1 -20741.124,E2 -20741.124} C_VEL
LIN {X 0,Y 213.737,Z 497.852,A -85,B 0,C 180,E1 -20743.67,E2 -20743.67} C_VEL
LIN {X 0,Y 213.801,Z 497.847,A -85,B 0,C 180,E1 -20746.351,E2 -20746.351} C_VEL
LIN {X 0,Y 213.788,Z 497.851,A -85,B 0,C 180,E1 -20749.12,E2 -20749.12} C_VEL
LIN {X 0,Y 213.745,Z 497.815,A -85,B 0,C 180,E1 -20753.716,E2 -20753.716} C_VEL
LIN {X 0,Y 213.788,Z 497.856,A -85,B 0,C 180,E1 -20758.727,E2 -20758.727} C_VEL
LIN {X 0,Y 213.819,Z 497.822,A -85,B 0,C 180,E1 -20762.606,E2 -20762.606} C_VEL
LIN {X 0,Y 213.846,Z 497.837,A -85,B 0,C 180,E1 -20766.956,E2 -20766.956} C_VEL
LIN {X 0,Y 213.887,Z 498.088,A -85,B 0,C 180,E1 -20771.072,E2 -20771.072} C_VEL
LIN {X 0,Y 214.202,Z 499.254,A -85,B 0,C 180,E1 -20771.379,E2 -20771.379} C_VEL
LIN {X 0,Y 220.592,Z 511.862,A -85,B 0,C 180,E1 -20772.744,E2 -20772.744} C_VEL
LIN {X 0,Y 228.316,Z 529.537,A -85,B 0,C 180,E1 -20774.345,E2 -20774.345} C_VEL
LIN {X 0,Y 228.871,Z 531.032,A -85,B 0,C 180,E1 -20774.463,E2 -20774.463} C_VEL
LIN {X 0,Y 227.92,Z 570.833,A -85,B 0,C 180,E1 -20775.722,E2 -20775.722} C_VEL
LIN {X 0,Y 227.644,Z 586.487,A -85,B 0,C 180,E1 -20776.354,E2 -20776.354} C_VEL
LIN {X 0,Y 226.97,Z 598.821,A -85,B 0,C 180,E1 -20777.18,E2 -20777.18} C_VEL
LIN {X 0,Y 226.019,Z 610.927,A -85,B 0,C 180,E1 -20778.342,E2 -20778.342} C_VEL
LIN {X 0,Y 224.685,Z 622.956,A -85,B 0,C 180,E1 -20779.869,E2 -20779.869} C_VEL
LIN {X 0,Y 223.085,Z 633.776,A -85,B 0,C 180,E1 -20781.625,E2 -20781.625} C_VEL
LIN {X 0,Y 221.52,Z 643.54,A -85,B 0,C 180,E1 -20783.628,E2 -20783.628} C_VEL
LIN {X 0,Y 219.89,Z 652.459,A -85,B 0,C 180,E1 -20785.879,E2 -20785.879} C_VEL
LIN {X 0,Y 218.245,Z 661.179,A -85,B 0,C 180,E1 -20788.619,E2 -20788.619} C_VEL
LIN {X 0,Y 216.849,Z 668.167,A -85,B 0,C 180,E1 -20791.396,E2 -20791.396} C_VEL
LIN {X 0,Y 215.61,Z 674.598,A -85,B 0,C 180,E1 -20794.677,E2 -20794.677} C_VEL
LIN {X 0,Y 214.899,Z 678.846,A -85,B 0,C 180,E1 -20797.52,E2 -20797.52} C_VEL
LIN {X 0,Y 214.494,Z 682.243,A -85,B 0,C 180,E1 -20800.595,E2 -20800.595} C_VEL
LIN {X 0,Y 214.431,Z 684.255,A -85,B 0,C 180,E1 -20803.266,E2 -20803.266} C_VEL
LIN {X 0,Y 214.56,Z 685.237,A -85,B 0,C 180,E1 -20805.194,E2 -20805.194} C_VEL
LIN {X 0,Y 215.303,Z 685.908,A -85,B 0,C 180,E1 -20808.806,E2 -20808.806} C_VEL
LIN {X 0,Y 215.987,Z 685.64,A -85,B 0,C 180,E1 -20810.976,E2 -20810.976} C_VEL
LIN {X 0,Y 216.771,Z 684.972,A -85,B 0,C 180,E1 -20812.899,E2 -20812.899} C_VEL
LIN {X 0,Y 218.284,Z 683.223,A -85,B 0,C 180,E1 -20815.645,E2 -20815.645} C_VEL
LIN {X 0,Y 220.998,Z 679.074,A -85,B 0,C 180,E1 -20819.536,E2 -20819.536} C_VEL
LIN {X 0,Y 223.479,Z 674.718,A -85,B 0,C 180,E1 -20822.321,E2 -20822.321} C_VEL
LIN {X 0,Y 226.318,Z 669.069,A -85,B 0,C 180,E1 -20825.067,E2 -20825.067} C_VEL
LIN {X 0,Y 229.511,Z 661.833,A -85,B 0,C 180,E1 -20827.769,E2 -20827.769} C_VEL
LIN {X 0,Y 233.167,Z 652.705,A -85,B 0,C 180,E1 -20830.397,E2 -20830.397} C_VEL
LIN {X 0,Y 236.283,Z 643.289,A -85,B 0,C 180,E1 -20832.53,E2 -20832.53} C_VEL
LIN {X 0,Y 239.082,Z 633.525,A -85,B 0,C 180,E1 -20834.282,E2 -20834.282} C_VEL
LIN {X 0,Y 241.847,Z 622.163,A -85,B 0,C 180,E1 -20835.881,E2 -20835.881} C_VEL
LIN {X 0,Y 243.953,Z 610.148,A -85,B 0,C 180,E1 -20837.204,E2 -20837.204} C_VEL
LIN {X 0,Y 245.472,Z 597.508,A -85,B 0,C 180,E1 -20838.239,E2 -20838.239} C_VEL
LIN {X 0,Y 245.632,Z 595.73,A -85,B 0,C 180,E1 -20838.365,E2 -20838.365} C_VEL
LIN {X 0,Y 242.545,Z 598.114,A -85,B 0,C 180,E1 -20838.805,E2 -20838.805} C_VEL
LIN {X 0,Y 239.684,Z 603.059,A -85,B 0,C 180,E1 -20838.948,E2 -20838.948} C_VEL
LIN {X 0,Y 236.696,Z 606.703,A -85,B 0,C 180,E1 -20839.215,E2 -20839.215} C_VEL
LIN {X 0,Y 233.451,Z 609.2,A -85,B 0,C 180,E1 -20839.666,E2 -20839.666} C_VEL
LIN {X 0,Y 230.639,Z 610.197,A -85,B 0,C 180,E1 -20840.216,E2 -20840.216} C_VEL
LIN {X 0,Y 228.253,Z 613.606,A -85,B 0,C 180,E1 -20840.336,E2 -20840.336} C_VEL
LIN {X 0,Y 226.542,Z 615.43,A -85,B 0,C 180,E1 -20840.508,E2 -20840.508} C_VEL
LIN {X 0,Y 224.941,Z 616.521,A -85,B 0,C 180,E1 -20840.752,E2 -20840.752} C_VEL
LIN {X 0,Y 223.589,Z 616.888,A -85,B 0,C 180,E1 -20841.05,E2 -20841.05} C_VEL
LIN {X 0,Y 222.492,Z 616.804,A -85,B 0,C 180,E1 -20841.441,E2 -20841.441} C_VEL
LIN {X 0,Y 221.943,Z 618.214,A -85,B 0,C 180,E1 -20841.869,E2 -20841.869} C_VEL
LIN {X 0,Y 221.677,Z 621.299,A -85,B 0,C 180,E1 -20842.144,E2 -20842.144} C_VEL
LIN {X 0,Y 220.557,Z 644.569,A -85,B 0,C 180,E1 -20843.312,E2 -20843.312} C_VEL
LIN {X 0,Y 219.583,Z 658.567,A -85,B 0,C 180,E1 -20844.402,E2 -20844.402} C_VEL
LIN {X 0,Y 218.513,Z 671.211,A -85,B 0,C 180,E1 -20845.748,E2 -20845.748} C_VEL
LIN {X 0,Y 217.082,Z 684.615,A -85,B 0,C 180,E1 -20847.618,E2 -20847.618} C_VEL
LIN {X 0,Y 215.737,Z 696.076,A -85,B 0,C 180,E1 -20849.674,E2 -20849.674} C_VEL
LIN {X 0,Y 214.49,Z 706.81,A -85,B 0,C 180,E1 -20852.059,E2 -20852.059} C_VEL
LIN {X 0,Y 213.416,Z 716.17,A -85,B 0,C 180,E1 -20854.654,E2 -20854.654} C_VEL
LIN {X 0,Y 212.599,Z 724.149,A -85,B 0,C 180,E1 -20857.369,E2 -20857.369} C_VEL
LIN {X 0,Y 212.011,Z 730.711,A -85,B 0,C 180,E1 -20860.137,E2 -20860.137} C_VEL
LIN {X 0,Y 211.688,Z 735.433,A -85,B 0,C 180,E1 -20862.615,E2 -20862.615} C_VEL
LIN {X 0,Y 211.504,Z 739.876,A -85,B 0,C 180,E1 -20865.57,E2 -20865.57} C_VEL
LIN {X 0,Y 211.57,Z 743.151,A -85,B 0,C 180,E1 -20868.504,E2 -20868.504} C_VEL
LIN {X 0,Y 211.853,Z 744.737,A -85,B 0,C 180,E1 -20870.453,E2 -20870.453} C_VEL
LIN {X 0,Y 212.461,Z 746.157,A -85,B 0,C 180,E1 -20872.938,E2 -20872.938} C_VEL
LIN {X 0,Y 213.598,Z 746.924,A -85,B 0,C 180,E1 -20876.228,E2 -20876.228} C_VEL
LIN {X 0,Y 215.729,Z 746.302,A -85,B 0,C 180,E1 -20880.001,E2 -20880.001} C_VEL
LIN {X 0,Y 218.214,Z 744.413,A -85,B 0,C 180,E1 -20883.179,E2 -20883.179} C_VEL
LIN {X 0,Y 221.426,Z 741.144,A -85,B 0,C 180,E1 -20886.379,E2 -20886.379} C_VEL
LIN {X 0,Y 224.706,Z 737.239,A -85,B 0,C 180,E1 -20888.998,E2 -20888.998} C_VEL
LIN {X 0,Y 228.447,Z 732.202,A -85,B 0,C 180,E1 -20891.536,E2 -20891.536} C_VEL
LIN {X 0,Y 229.838,Z 730.181,A -85,B 0,C 180,E1 -20892.4,E2 -20892.4} C_VEL
LIN {X 0,Y 231.282,Z 727.36,A -85,B 0,C 180,E1 -20893.642,E2 -20893.642} C_VEL
LIN {X 0,Y 232.375,Z 722.833,A -85,B 0,C 180,E1 -20895.812,E2 -20895.812} C_VEL
LIN {X 0,Y 233.668,Z 717.792,A -85,B 0,C 180,E1 -20897.873,E2 -20897.873} C_VEL
LIN {X 0,Y 235.347,Z 714.147,A -85,B 0,C 180,E1 -20898.921,E2 -20898.921} C_VEL
LIN {X 0,Y 240.548,Z 704.152,A -85,B 0,C 180,E1 -20901.011,E2 -20901.011} C_VEL
LIN {X 0,Y 245.665,Z 692.823,A -85,B 0,C 180,E1 -20902.84,E2 -20902.84} C_VEL
LIN {X 0,Y 250.026,Z 681.318,A -85,B 0,C 180,E1 -20904.274,E2 -20904.274} C_VEL
LIN {X 0,Y 254.21,Z 667.601,A -85,B 0,C 180,E1 -20905.594,E2 -20905.594} C_VEL
LIN {X 0,Y 257.476,Z 653.847,A -85,B 0,C 180,E1 -20906.55,E2 -20906.55} C_VEL
LIN {X 0,Y 260.664,Z 635.193,A -85,B 0,C 180,E1 -20907.428,E2 -20907.428} C_VEL
LIN {X 0,Y 268.35,Z 590.01,A -85,B 0,C 180,E1 -20909.295,E2 -20909.295} C_VEL
LIN {X 0,Y 266.847,Z 584.876,A -85,B 0,C 180,E1 -20911.377,E2 -20911.377} C_VEL
LIN {X 0,Y 265.885,Z 581.947,A -85,B 0,C 180,E1 -20913.08,E2 -20913.08} C_VEL
LIN {X 0,Y 265.057,Z 579.441,A -85,B 0,C 180,E1 -20915.338,E2 -20915.338} C_VEL
LIN {X 0,Y 264.755,Z 578.251,A -85,B 0,C 180,E1 -20917.629,E2 -20917.629} C_VEL
LIN {X 0,Y 265.272,Z 578.373,A -85,B 0,C 180,E1 -20920.722,E2 -20920.722} C_VEL
LIN {X 0,Y 266.413,Z 579.943,A -85,B 0,C 180,E1 -20923.11,E2 -20923.11} C_VEL
LIN {X 0,Y 266.715,Z 580.556,A -85,B 0,C 180,E1 -20923.589,E2 -20923.589} C_VEL
LIN {X 0,Y 267.007,Z 585.619,A -85,B 0,C 180,E1 -20925.035,E2 -20925.035} C_VEL
LIN {X 0,Y 265.895,Z 598.144,A -85,B 0,C 180,E1 -20926.416,E2 -20926.416} C_VEL
LIN {X 0,Y 264.767,Z 609.276,A -85,B 0,C 180,E1 -20927.453,E2 -20927.453} C_VEL
LIN {X 0,Y 263.384,Z 620.363,A -85,B 0,C 180,E1 -20928.218,E2 -20928.218} C_VEL
LIN {X 0,Y 256.053,Z 663.709,A -85,B 0,C 180,E1 -20930.087,E2 -20930.087} C_VEL
LIN {X 0,Y 252.311,Z 678.504,A -85,B 0,C 180,E1 -20930.931,E2 -20930.931} C_VEL
LIN {X 0,Y 248.235,Z 691.457,A -85,B 0,C 180,E1 -20931.988,E2 -20931.988} C_VEL
LIN {X 0,Y 243.688,Z 703.28,A -85,B 0,C 180,E1 -20933.239,E2 -20933.239} C_VEL
LIN {X 0,Y 238.331,Z 715.143,A -85,B 0,C 180,E1 -20934.896,E2 -20934.896} C_VEL
LIN {X 0,Y 233.47,Z 724.981,A -85,B 0,C 180,E1 -20936.673,E2 -20936.673} C_VEL
LIN {X 0,Y 228.008,Z 734.667,A -85,B 0,C 180,E1 -20938.913,E2 -20938.913} C_VEL
LIN {X 0,Y 223.06,Z 742.677,A -85,B 0,C 180,E1 -20941.28,E2 -20941.28} C_VEL
LIN {X 0,Y 219.359,Z 748.272,A -85,B 0,C 180,E1 -20943.347,E2 -20943.347} C_VEL
LIN {X 0,Y 215.187,Z 754.222,A -85,B 0,C 180,E1 -20946.133,E2 -20946.133} C_VEL
LIN {X 0,Y 212.199,Z 758.326,A -85,B 0,C 180,E1 -20948.631,E2 -20948.631} C_VEL
LIN {X 0,Y 209.62,Z 761.816,A -85,B 0,C 180,E1 -20951.424,E2 -20951.424} C_VEL
LIN {X 0,Y 207.4,Z 764.383,A -85,B 0,C 180,E1 -20954.268,E2 -20954.268} C_VEL
LIN {X 0,Y 205.579,Z 766.444,A -85,B 0,C 180,E1 -20958.16,E2 -20958.16} C_VEL
LIN {X 0,Y 205.051,Z 766.9,A -85,B 0,C 180,E1 -20960.129,E2 -20960.129} C_VEL
LIN {X 0,Y 204.683,Z 766.581,A -85,B 0,C 180,E1 -20964.084,E2 -20964.084} C_VEL
LIN {X 0,Y 204.779,Z 765.824,A -85,B 0,C 180,E1 -20966.061,E2 -20966.061} C_VEL
LIN {X 0,Y 204.99,Z 764.658,A -85,B 0,C 180,E1 -20968.032,E2 -20968.032} C_VEL
LIN {X 0,Y 205.385,Z 763.03,A -85,B 0,C 180,E1 -20969.997,E2 -20969.997} C_VEL
LIN {X 0,Y 205.193,Z 759.548,A -85,B 0,C 180,E1 -20972.942,E2 -20972.942} C_VEL
LIN {X 0,Y 205.209,Z 754.834,A -85,B 0,C 180,E1 -20975.894,E2 -20975.894} C_VEL
LIN {X 0,Y 205.363,Z 748.676,A -85,B 0,C 180,E1 -20978.855,E2 -20978.855} C_VEL
LIN {X 0,Y 205.785,Z 740.854,A -85,B 0,C 180,E1 -20981.821,E2 -20981.821} C_VEL
LIN {X 0,Y 206.508,Z 732.774,A -85,B 0,C 180,E1 -20984.281,E2 -20984.281} C_VEL
LIN {X 0,Y 207.561,Z 722.944,A -85,B 0,C 180,E1 -20986.723,E2 -20986.723} C_VEL
LIN {X 0,Y 208.977,Z 710.867,A -85,B 0,C 180,E1 -20989.138,E2 -20989.138} C_VEL
LIN {X 0,Y 210.752,Z 700.647,A -85,B 0,C 180,E1 -20991.773,E2 -20991.773} C_VEL
LIN {X 0,Y 212.637,Z 690.319,A -85,B 0,C 180,E1 -20993.88,E2 -20993.88} C_VEL
LIN {X 0,Y 214.842,Z 678.939,A -85,B 0,C 180,E1 -20995.682,E2 -20995.682} C_VEL
LIN {X 0,Y 216.683,Z 667.109,A -85,B 0,C 180,E1 -20997.133,E2 -20997.133} C_VEL
LIN {X 0,Y 218.244,Z 654.213,A -85,B 0,C 180,E1 -20998.289,E2 -20998.289} C_VEL
LIN {X 0,Y 219.336,Z 641.174,A -85,B 0,C 180,E1 -20999.075,E2 -20999.075} C_VEL
LIN {X 0,Y 220.277,Z 615.238,A -85,B 0,C 180,E1 -20999.966,E2 -20999.966} C_VEL
LIN {X 0,Y 220.227,Z 606.731,A -85,B 0,C 180,E1 -21000.272,E2 -21000.272} C_VEL
LIN {X 0,Y 215.956,Z 547.394,A -85,B 0,C 180,E1 -21002.936,E2 -21002.936} C_VEL
LIN {X 0,Y 214.212,Z 530.993,A -85,B 0,C 180,E1 -21003.768,E2 -21003.768} C_VEL
LIN {X 0,Y 213.346,Z 528.217,A -85,B 0,C 180,E1 -21004.052,E2 -21004.052} C_VEL
LIN {X 0,Y 211.242,Z 517.598,A -85,B 0,C 180,E1 -21007.799,E2 -21007.799} C_VEL
LIN {X 0,Y 208.584,Z 506.197,A -85,B 0,C 180,E1 -21012.16,E2 -21012.16} C_VEL
LIN {X 0,Y 206.695,Z 498.846,A -85,B 0,C 180,E1 -21015.251,E2 -21015.251} C_VEL
LIN {X 0,Y 206.652,Z 498.736,A -85,B 0,C 180,E1 -21019.746,E2 -21019.746} C_VEL
LIN {X 0,Y 206.69,Z 498.724,A -85,B 0,C 180,E1 -21024.686,E2 -21024.686} C_VEL
LIN {X 0,Y 206.697,Z 498.736,A -85,B 0,C 180,E1 -21029.334,E2 -21029.334} C_VEL
LIN {X 0,Y 206.723,Z 498.723,A -85,B 0,C 180,E1 -21033.77,E2 -21033.77} C_VEL
LIN {X 0,Y 206.747,Z 498.725,A -85,B 0,C 180,E1 -21038.041,E2 -21038.041} C_VEL
LIN {X 0,Y 206.862,Z 498.708,A -85,B 0,C 180,E1 -21042.195,E2 -21042.195} C_VEL
LIN {X 0,Y 206.902,Z 498.706,A -85,B 0,C 180,E1 -21046.244,E2 -21046.244} C_VEL
LIN {X 0,Y 207.094,Z 498.669,A -85,B 0,C 180,E1 -21050.23,E2 -21050.23} C_VEL
LIN {X 0,Y 207.166,Z 498.674,A -85,B 0,C 180,E1 -21052.2,E2 -21052.2} C_VEL
LIN {X 0,Y 207.369,Z 498.629,A -85,B 0,C 180,E1 -21058.057,E2 -21058.057} C_VEL
LIN {X 0,Y 207.502,Z 498.617,A -85,B 0,C 180,E1 -21059.999,E2 -21059.999} C_VEL
LIN {X 0,Y 207.37,Z 498.647,A -85,B 0,C 180,E1 -21061.941,E2 -21061.941} C_VEL
LIN {X 0,Y 207.155,Z 498.658,A -85,B 0,C 180,E1 -21067.799,E2 -21067.799} C_VEL
LIN {X 0,Y 206.969,Z 498.696,A -85,B 0,C 180,E1 -21071.755,E2 -21071.755} C_VEL
LIN {X 0,Y 206.855,Z 498.715,A -85,B 0,C 180,E1 -21075.771,E2 -21075.771} C_VEL
LIN {X 0,Y 206.771,Z 498.703,A -85,B 0,C 180,E1 -21079.87,E2 -21079.87} C_VEL
LIN {X 0,Y 206.751,Z 498.729,A -85,B 0,C 180,E1 -21084.073,E2 -21084.073} C_VEL
LIN {X 0,Y 206.732,Z 498.711,A -85,B 0,C 180,E1 -21088.42,E2 -21088.42} C_VEL
LIN {X 0,Y 206.69,Z 498.74,A -85,B 0,C 180,E1 -21092.958,E2 -21092.958} C_VEL
LIN {X 0,Y 206.669,Z 498.723,A -85,B 0,C 180,E1 -21097.741,E2 -21097.741} C_VEL
LIN {X 0,Y 206.645,Z 498.744,A -85,B 0,C 180,E1 -21101.569,E2 -21101.569} C_VEL
LIN {X 0,Y 206.698,Z 498.726,A -85,B 0,C 180,E1 -21105.562,E2 -21105.562} C_VEL
LIN {X 0,Y 206.718,Z 498.729,A -85,B 0,C 180,E1 -21109.767,E2 -21109.767} C_VEL
LIN {X 0,Y 206.716,Z 498.695,A -85,B 0,C 180,E1 -21112.272,E2 -21112.272} C_VEL
LIN {X 0,Y 206.701,Z 498.731,A -85,B 0,C 180,E1 -21117.047,E2 -21117.047} C_VEL
LIN {X 0,Y 206.759,Z 498.699,A -85,B 0,C 180,E1 -21122.099,E2 -21122.099} C_VEL
LIN {X 0,Y 206.779,Z 498.72,A -85,B 0,C 180,E1 -21126.587,E2 -21126.587} C_VEL
LIN {X 0,Y 206.808,Z 498.932,A -85,B 0,C 180,E1 -21130.008,E2 -21130.008} C_VEL
LIN {X 0,Y 207.06,Z 499.988,A -85,B 0,C 180,E1 -21130.337,E2 -21130.337} C_VEL
LIN {X 0,Y 214.491,Z 514.456,A -85,B 0,C 180,E1 -21132.009,E2 -21132.009} C_VEL
LIN {X 0,Y 221.851,Z 531.331,A -85,B 0,C 180,E1 -21133.608,E2 -21133.608} C_VEL
LIN {X 0,Y 222.43,Z 533.132,A -85,B 0,C 180,E1 -21133.746,E2 -21133.746} C_VEL
LIN {X 0,Y 221.456,Z 572.091,A -85,B 0,C 180,E1 -21135.013,E2 -21135.013} C_VEL
LIN {X 0,Y 221.167,Z 586.995,A -85,B 0,C 180,E1 -21135.629,E2 -21135.629} C_VEL
LIN {X 0,Y 220.534,Z 598.673,A -85,B 0,C 180,E1 -21136.41,E2 -21136.41} C_VEL
LIN {X 0,Y 219.584,Z 610.429,A -85,B 0,C 180,E1 -21137.527,E2 -21137.527} C_VEL
LIN {X 0,Y 218.196,Z 622.749,A -85,B 0,C 180,E1 -21139.095,E2 -21139.095} C_VEL
LIN {X 0,Y 216.543,Z 633.818,A -85,B 0,C 180,E1 -21140.9,E2 -21140.9} C_VEL
LIN {X 0,Y 214.896,Z 643.776,A -85,B 0,C 180,E1 -21142.959,E2 -21142.959} C_VEL
LIN {X 0,Y 213.181,Z 652.816,A -85,B 0,C 180,E1 -21145.276,E2 -21145.276} C_VEL
LIN {X 0,Y 211.428,Z 661.648,A -85,B 0,C 180,E1 -21148.098,E2 -21148.098} C_VEL
LIN {X 0,Y 209.972,Z 668.76,A -85,B 0,C 180,E1 -21150.962,E2 -21150.962} C_VEL
